// TwinCAT 3 PLC project BROTLib
// Title: BROTLib
// Company: BROT
// ProjectVersion: 0.6.1
// ProgramVersion: 3.1.4026.16
// libraries:
//   AstroBROT, * (BROT)
//   Tc2_Math, * (Beckhoff Automation GmbH)
//   Tc2_MC2, * (Beckhoff Automation GmbH)
//   Tc2_MC2_Drive, * (Beckhoff Automation GmbH)
//   Tc2_NC, * (Beckhoff Automation GmbH)
//   Tc2_Standard, * (Beckhoff Automation GmbH)
//   Tc2_System, * (Beckhoff Automation GmbH)
//   Tc2_Utilities, * (Beckhoff Automation GmbH)
//   Tc3_IotBase, * (Beckhoff Automation GmbH)
//   Tc3_IotCommunicator, * (Beckhoff Automation GmbH)
// project tree:
//   Interfaces/ I_AltAzTelescope.TcIO, I_Axis.TcIO, I_BaseAxis.TcIO, I_Brake.TcIO, I_Dome.TcIO, I_Filter.TcIO, I_Focus.TcIO, I_Hydraulics.TcIO, I_MirrorCovers.TcIO, I_Nasmyth.TcIO, I_RaDecTelescope.TcIO (not stored), I_Roof.TcIO, I_Telescope.TcIO
//   DUTs/ E_Blink.TcDUT, E_DomeRotationState.TcDUT, E_Horn.TcDUT, E_RoofState.TcDUT, E_TCSCommand.TcDUT, E_TelescopeMode.TcDUT, ST_AltAzCoordinate.TcDUT, ST_InfoDataConnection.TcDUT (not stored), ST_InfoDataFB.TcDUT (not stored), ST_InfoDataGroup.TcDUT (not stored), ST_RaDecCoordinate.TcDUT
//   GVLs/ GVL_Math.TcGVL, Global_Version.TcGVL
//   POUs/Comm/ FB_Comm_MQTT.TcPOU, FB_Comm_MQTT_Influx.TcPOU, F_EscapeInfluxString.TcPOU, F_EscapeInfluxTag.TcPOU, F_InfluxFieldValue.TcPOU, F_InfluxTimestamp.TcPOU, F_IsNumericValue.TcPOU, F_TruncateInfluxEscaped.TcPOU, I_Comm.TcIO
//   POUs/Debug/ FB_InfoConnection.TcPOU, FB_InfoEStop.TcPOU, FB_InfoGroup.TcPOU
//   POUs/ FB_AstroClock.TcPOU, FB_AstroClockSync.TcPOU, F_SetpointEnableExecute.TcPOU, FB_Axis.TcPOU, FB_BaseAxis.TcPOU, FB_BLINK.TcPOU, FB_ButtonEnable.TcPOU, FB_EventLog.TcPOU, FB_Horn.TcPOU, FB_InfluxMessage.TcPOU, FB_TONTP.TcPOU, F_YREAL.TcPOU, NCError_TO_STRING.TcPOU
//   POUs/Pointing/ FB_PointingModelForward.TcPOU, FB_PointingModelInversion.TcPOU
//   POUs/Tracking/ F_Azimuthvelocity.TcPOU, F_DerotatorPosition2.TcPOU, F_Derotatorvelocity.TcPOU, F_Elevationvelocity.TcPOU
//   Telescope/ FB_AltAzTelescopeControl.TcPOU, FB_BaseTelescopeControl.TcPOU, FB_RaDecTelescopeControl.TcPOU, ST_TelescopeConfig.TcDUT

// ---- DUTs/E_Blink.TcDUT
{attribute 'qualified_only'}
{attribute 'strict'}
TYPE E_Blink :
(
	off := 0,
	slow,
	fast,
	short,
	long,
	on
);
END_TYPE

// ---- DUTs/E_DomeRotationState.TcDUT
{attribute 'qualified_only'}
{attribute 'strict'}
TYPE E_DomeRotationState :
(
	idle  := 0,
	parked	:= 1,
	slewing := 2,
	error	:= 3,
	unknown := 4
);
END_TYPE

// ---- DUTs/E_Horn.TcDUT
{attribute 'qualified_only'}
{attribute 'strict'}
TYPE E_Horn :
(
	off := 0,
	beep,
	short,
	long
);
END_TYPE

// ---- DUTs/E_RoofState.TcDUT
{attribute 'qualified_only'}
{attribute 'strict'}
TYPE E_RoofState :
(
	closed := 0,
	opened := 1,
	opening := 2,
	closing := 3,
	stopped := 4,
	error := 5,
	unknown := 6
);
END_TYPE

// ---- DUTs/E_TCSCommand.TcDUT
{attribute 'qualified_only'}
{attribute 'strict'}
TYPE E_TCSCommand :
(
	no_command := 0,
	gohome,
	park,
	track,
	goto,
	stop,
	slew,
	poweron
);
END_TYPE

// ---- DUTs/E_TelescopeMode.TcDUT
{attribute 'qualified_only'}
{attribute 'strict'}
TYPE E_TelescopeMode :
(
	off := 0,
	manual := 1,
	automatic := 2
);
END_TYPE

// ---- DUTs/ST_AltAzCoordinate.TcDUT
TYPE ST_AltAzCoordinate :
STRUCT
	Altitude : LREAL;
	Azimuth  : LREAL;
END_STRUCT
END_TYPE

// ---- DUTs/ST_RaDecCoordinate.TcDUT
TYPE ST_RaDecCoordinate :
STRUCT
	RightAscension  : LREAL;
	Declination : LREAL;
END_STRUCT
END_TYPE

// ---- Telescope/ST_TelescopeConfig.TcDUT
TYPE ST_TelescopeConfig :
STRUCT
	// location
	longitude			: LREAL; // telescope site longitude
	latitude			: LREAL; // telescope site latitude
	altitude			: LREAL; // telescope site height above sea level: estimated
	
	// park position
	elevationPark		: LREAL;
	azimuthPark			: LREAL;
	derotatorPark		: LREAL;
	focusPark			: LREAL;

	// home position
	elevationHome		: LREAL;
	azimuthHome			: LREAL;
	derotatorHome		: LREAL;
	
	// information about telescope
	name				: STRING;
	diameter			: LREAL;
	cabinet				: STRING;
	manufacturer		: STRING;
	
	// and about the mount
	mountOptions		: STRING;
	mount				: STRING;	
END_STRUCT
END_TYPE

// ---- GVLs/GVL_Math.TcGVL
{attribute 'qualified_only'}
VAR_GLOBAL CONSTANT
	LREAL_MIN			: LREAL :=  -1.7976931348623157E+308; // https://infosys.beckhoff.com/index.php?content=../content/1031/tc3_plc_intro/2529405067.html&id=
	// literal values (PI/180 and 180/PI), not PI-based expressions: PI is not initialised yet when these
	// constants are, which fails the build ("uninitialized variable PI is used for initialization")
	d2r					: LREAL := 0.017453292519943295;
	r2d					: LREAL := 57.29577951308232;
	// Earth's mean sidereal angular rate, deg/s (360 deg / 86164.0905 s mean sidereal day); was previously
	// copy-pasted into three tracking functions, and separately (re-derived slightly differently, as
	// 360/86164.099, ~0.005 arcsec/hour off) as the unused FB_BaseTelescopeControl.fSiderialVelocity
	Omega				: LREAL := 4.178074605556E-3;
END_VAR

// ---- GVLs/Global_Version.TcGVL
{attribute 'qualified_only'}
VAR_GLOBAL CONSTANT
	// Mirrors Beckhoff's own Global_Version.stLibVersion_* pattern (see ST_LibVersion),
	// which only covers Tc2_*/Tc3_* library references, not custom ones -- until now: this
	// GVL uses Beckhoff's own naming exactly, so it merges into a consumer's Global_Version.
	// Kept in sync with <ProjectVersion> in BROTLib.plcproj at release time.
	stLibVersion_BROTLib : ST_LibVersion := (
		iMajor := 0,
		iMinor := 6,
		iBuild := 1,
		iRevision := 0,
		nFlags := 1,
		sVersion := '0.6.1'
	);
END_VAR

// ---- Interfaces/I_AltAzTelescope.TcIO
INTERFACE I_AltAzTelescope EXTENDS I_Telescope

PROPERTY AltitudeOffset : LREAL
GET
END_GET
SET
END_SET
END_PROPERTY

PROPERTY AzimuthOffset : LREAL
GET
END_GET
SET
END_SET
END_PROPERTY

PROPERTY DerotatorOffset : LREAL
GET
END_GET
SET
END_SET
END_PROPERTY

PROPERTY Dut1 : LREAL
GET
END_GET
SET
END_SET
END_PROPERTY

END_INTERFACE

// ---- Interfaces/I_Axis.TcIO
INTERFACE I_Axis EXTENDS I_BaseAxis

PROPERTY ActualPosition : LREAL
GET
END_GET
SET
END_SET
END_PROPERTY

PROPERTY isTracking : BOOL
GET
END_GET
END_PROPERTY

PROPERTY MoveAxis : BOOL
GET
END_GET
SET
END_SET
END_PROPERTY

PROPERTY MoveDone : BOOL
GET
END_GET
END_PROPERTY

PROPERTY SlewTime : LREAL
GET
END_GET
END_PROPERTY

PROPERTY StopAxis : BOOL
GET
END_GET
SET
END_SET
END_PROPERTY

PROPERTY Tracking : BOOL
GET
END_GET
SET
END_SET
END_PROPERTY

END_INTERFACE

// ---- Interfaces/I_BaseAxis.TcIO
INTERFACE I_BaseAxis

PROPERTY ActualPosition : LREAL
GET
END_GET
SET
END_SET
END_PROPERTY

PROPERTY Busy : BOOL
GET
END_GET
END_PROPERTY

PROPERTY Calibrated : BOOL
GET
END_GET
END_PROPERTY

PROPERTY Enable : BOOL
GET
END_GET
SET
END_SET
END_PROPERTY

PROPERTY Error : BOOL
GET
END_GET
END_PROPERTY

PROPERTY ErrorID : UDINT
GET
END_GET
END_PROPERTY

PROPERTY HomeAxis : BOOL
GET
END_GET
SET
END_SET
END_PROPERTY

PROPERTY InNegLimit : BOOL
GET
END_GET
END_PROPERTY

PROPERTY InPosLimit : BOOL
GET
END_GET
END_PROPERTY

PROPERTY MoveNeg : BOOL
GET
END_GET
SET
END_SET
END_PROPERTY

PROPERTY MovePos : BOOL
GET
END_GET
SET
END_SET
END_PROPERTY

PROPERTY Position : LREAL
GET
END_GET
SET
END_SET
END_PROPERTY

PROPERTY Ready : BOOL
GET
END_GET
END_PROPERTY

METHOD Reset : BOOL
VAR_INPUT
END_VAR
END_METHOD

PROPERTY Velocity : LREAL
GET
END_GET
SET
END_SET
END_PROPERTY

END_INTERFACE

// ---- Interfaces/I_Brake.TcIO
INTERFACE I_Brake

PROPERTY BrakeOpen : BOOL
GET
END_GET
END_PROPERTY

METHOD CloseBrake : BOOL
VAR_INPUT
END_VAR
END_METHOD

METHOD OpenBrake : BOOL
VAR_INPUT
END_VAR
END_METHOD

END_INTERFACE

// ---- Interfaces/I_Dome.TcIO
INTERFACE I_Dome

PROPERTY Capabilities : INT
GET
END_GET
END_PROPERTY

METHOD Close : BOOL
VAR_INPUT
END_VAR
END_METHOD

PROPERTY Error : BOOL
GET
END_GET
END_PROPERTY

PROPERTY ErrorID : UDINT
GET
END_GET
END_PROPERTY

METHOD Open : BOOL
VAR_INPUT
END_VAR
END_METHOD

METHOD Park : BOOL
VAR_INPUT
END_VAR
END_METHOD

PROPERTY Parked : BOOL
GET
END_GET
END_PROPERTY

PROPERTY Position : LREAL
GET
END_GET
SET
END_SET
END_PROPERTY

METHOD Reset : BOOL
VAR_INPUT
END_VAR
END_METHOD

PROPERTY RotState : E_DomeRotationState
GET
END_GET
END_PROPERTY

PROPERTY ShutterState : E_RoofState
GET
END_GET
SET
END_SET
END_PROPERTY

METHOD Stop : BOOL
VAR_INPUT
END_VAR
END_METHOD

METHOD StopTrack : BOOL
VAR_INPUT
END_VAR
END_METHOD

METHOD Track : BOOL
VAR_INPUT
END_VAR
END_METHOD

PROPERTY Tracking : BOOL
GET
END_GET
END_PROPERTY

END_INTERFACE

// ---- Interfaces/I_Filter.TcIO
INTERFACE I_Filter

METHOD SetFilter : BOOL
VAR_INPUT
	FilterPos	: USINT;
END_VAR
END_METHOD

END_INTERFACE

// ---- Interfaces/I_Focus.TcIO
INTERFACE I_Focus EXTENDS I_BaseAxis

END_INTERFACE

// ---- Interfaces/I_Hydraulics.TcIO
INTERFACE I_Hydraulics

PROPERTY Enable : BOOL
GET
END_GET
SET
END_SET
END_PROPERTY

PROPERTY Error : BOOL
GET
END_GET
END_PROPERTY

PROPERTY ManualStartSuction : BOOL
GET
END_GET
SET
END_SET
END_PROPERTY

PROPERTY ManualStopPump : BOOL
GET
END_GET
SET
END_SET
END_PROPERTY

PROPERTY OilPressureOK : BOOL
GET
END_GET
END_PROPERTY

PROPERTY PumpRunning : BOOL
GET
END_GET
END_PROPERTY

METHOD Reset : BOOL
VAR_INPUT
END_VAR
END_METHOD

PROPERTY SuctionRunning : BOOL
GET
END_GET
END_PROPERTY

END_INTERFACE

// ---- Interfaces/I_MirrorCovers.TcIO
INTERFACE I_MirrorCovers

METHOD Close : BOOL
VAR_INPUT
END_VAR
END_METHOD

PROPERTY Closed : BOOL
GET
END_GET
END_PROPERTY

PROPERTY Error : BOOL
GET
END_GET
END_PROPERTY

METHOD Open : BOOL
VAR_INPUT
END_VAR
END_METHOD

PROPERTY Opened : BOOL
GET
END_GET
END_PROPERTY

METHOD Reset : BOOL
VAR_INPUT
END_VAR
END_METHOD

END_INTERFACE

// ---- Interfaces/I_Nasmyth.TcIO
INTERFACE I_Nasmyth

METHOD SetNasmyth : BOOL
VAR_INPUT
	Port	: INT;
END_VAR
END_METHOD

END_INTERFACE

// ---- Interfaces/I_Roof.TcIO
INTERFACE I_Roof

METHOD Close : BOOL
VAR_INPUT
END_VAR
END_METHOD

METHOD Open : BOOL
VAR_INPUT
END_VAR
END_METHOD

METHOD Reset : BOOL
VAR_INPUT
END_VAR
END_METHOD

PROPERTY State : E_RoofState
GET
END_GET
END_PROPERTY

METHOD Stop : BOOL
VAR_INPUT
END_VAR
END_METHOD

END_INTERFACE

// ---- Interfaces/I_Telescope.TcIO
INTERFACE I_Telescope

PROPERTY Altitude : LREAL
GET
END_GET
END_PROPERTY

PROPERTY Azimuth : LREAL
GET
END_GET
END_PROPERTY

PROPERTY CoverAutoOpen : BOOL
GET
END_GET
SET
END_SET
END_PROPERTY

PROPERTY Declination : LREAL
GET
END_GET
END_PROPERTY

METHOD ABSTRACT Home : BOOL
VAR_INPUT
END_VAR
END_METHOD

METHOD Init : BOOL
VAR_INPUT
END_VAR
END_METHOD

METHOD ABSTRACT Park : BOOL
VAR_INPUT
END_VAR
END_METHOD

METHOD Reset : BOOL
VAR_INPUT
END_VAR
END_METHOD

PROPERTY RightAscension : LREAL
GET
END_GET
END_PROPERTY

METHOD Slew : BOOL
VAR_INPUT
	fAzimuth		: LREAL;
	fAltitude		: LREAL;
END_VAR
END_METHOD

METHOD Stop : BOOL
VAR_INPUT
END_VAR
END_METHOD

METHOD Track : BOOL
VAR_INPUT
	fRightAscension	: LREAL;
	fDeclination	: LREAL;
END_VAR
END_METHOD

END_INTERFACE

// ---- POUs/Comm/I_Comm.TcIO
INTERFACE I_Comm

METHOD Publish : BOOL
VAR_INPUT
	domain			: STRING(255) := 'environment';
	location		: STRING(255) := 'roof';
	parameter		: STRING(255);
	value			: STRING(255);	
END_VAR
VAR_OUTPUT
	published	: BOOL;
END_VAR
END_METHOD

METHOD PublishLog : BOOL
VAR_INPUT
	level		: STRING(255) := 'INFO';
	message		: STRING(255);	
END_VAR
VAR_OUTPUT
	published	: BOOL;
END_VAR
END_METHOD

END_INTERFACE

// ---- Telescope/FB_BaseTelescopeControl.TcPOU
FUNCTION_BLOCK ABSTRACT FB_BaseTelescopeControl IMPLEMENTS I_Telescope
VAR_INPUT
(*
TCS interface section, modeled on an external TCS spec kept as a private internal reference
(not linked here -- this repo is public; ask internally for the spec if you need it). See
specs/design/telescope-telemetry-publish-chain.md for what's actually confirmed about the
on-wire format from tracing the code, since the spec itself isn't accessible from here.
*)
	bPower				: BOOL;		// true: Power on
	bGoHome				: BOOL;		// true: go to home position, unset track/goto if active
	bPark				: BOOL;		// boolean, true: go into park position, ready to stow telescope, unset track/goto
	bTrack				: BOOL;		// boolean, TRUE: MOVE telescope TO last ra/de AND start tracking. Set 'goto' TO FALSE, IF TRUE. FALSE: Stop tracking as soon as possible
	bGoto				: BOOL;		// boolean, TRUE: MOVE telescope TO tau/de AND stop there. Set track TO FALSE, IF TRUE. FALSE: no effect.)	
	bSlew				: BOOL;		// move the telescope to a given az-alt position
	bStop				: BOOL;		// boolean, TRUE: Stop motion OF telescope immediately, set goto AND track TO FALSE. FALSE: Allow motion OF telescope again via track/goto).	
	bReset				: BOOL;		// initiates reset on all axis
	bAutoTrack			: BOOL := TRUE;	// automatic tracking after goto
	bCoverAutoOpen		: BOOL := TRUE;	// automatically open the mirror covers on Init/PowerOn
	// catalog/mean right ascension (ICRS/J2000), degrees, double -- fed straight into AstroBROT's
	// FB_EQ2HOR with precess/nutate/aberration all at their default TRUE, which only makes sense
	// for mean/catalog input (feeding it an already-apparent position would double-correct it);
	// MONETcommon's own telemetry independently re-publishes this same value as *_RA_ICRS (#22)
	fRightAscension		: LREAL :=  0.0;
	// catalog/mean declination (ICRS/J2000), degrees, double -- see fRightAscension
	fDeclination		: LREAL :=  0.0;
	fElevation			: LREAL :=  0.0;	// desired elevation of the telescope pointing
	fAzimuth			: LREAL :=  0.0;	// desired azimut of the telescope pointing
	fTimeOffset			: LREAL := 0.0;		// absolute offset for time
	fHorizon			: LREAL := 1.0;		// ELEVATION below which value the telescope will not go
	
	// TRUE while the E-stop is triggered. The caller must connect it to its safety handling (MONETS/MONETN MAIN:
	// SafetyHandling.estop); left unconnected, the E-stop is never reported as STATUS.GLOBAL = 1 (#10).
	bEstopTriggered		: BOOL	:= FALSE;
	bMainReady			: BOOL	:= TRUE;
	
	telescopeConfig		: ST_TelescopeConfig;
END_VAR
VAR
	fbComm 				: I_Comm;
	
	TCS_command			: E_TCSCommand;	// actual command from the TCS
	// fJd/fLst are published by _PublishTelemetry, but this block never sets them or calls fbTime: the derived
	// block must (MONETcommon's FB_MonetTelescopeControl does, gated on fbTime.bValid). Otherwise both read 0 (#10).
	fJd					: LREAL;	// current Julian Date calculated from system time
	fLst				: LREAL;	// local siderial time calculated from Julian date in hours
	fElevationCalc		: LREAL;	// elevation calulated when ra and dec are set by TCS 
	fAzimuthCalc		: LREAL;	// azimuth calulated when ra and dec are set by TCS
	fHourAngle			: LREAL;	// hourangle when ra and dec are set by TCS
	
	fRightAscensionCalc	: LREAL;	// right ascension calulated when azimuth and elevation are set by TCS
	fDeclinationCalc	: LREAL;	// declination calulated when azimuth and elevation are set by TCS
	fHourAngleCalc		: LREAL;	// hour angle azimuth and elevation are set by TCS
	
	fbTime				: FB_AstroClock;	// precise astronomical	time
	
	rtrigReset			: R_TRIG;
	bInterrupted		: BOOL;		// If a command is interruped by one with more presedence, the interrupted needs to reset its stage
	
	bPowerFailure		: BOOL;		// triggers power-failure event
	tpPowerOnWarning	: TP;		// triggers power warning
	tonPowerTimeout		: TON;		// power on timeout
	tonCommandTimeout	: TON;		// command timeout
	tonTrackingDelay	: TON;		// tracking delay
	
	TCSpowerEvent,
	TCSgohomeEvent,
	TCSparkEvent,
	TCSgotoEvent,
	TCStrackEvent,
	TCSstopEvent,
	TCStargetHorizonEvent,
	TCSaltitudeEvent,
	TCSnearPoleEvent,
	TCSreadyEvent,
	TCSCTOEvent			: FB_Eventlog;
	tonMQTTTimer 			: TON := (PT:=T#5S);
	// the 7 INFO/CONFIG fields never change at runtime; republishing them on the fast 1-5s
	// telemetry cadence is wasted traffic, so they get their own much slower timer instead
	tonStaticTelemetryTimer	: TON := (PT:=T#30S);
	bStaticTelemetrySent	: BOOL;	// forces one immediate publish on the first cycle
END_VAR
VAR_OUTPUT
	bReady				: BOOL;		// TRUE, IF telescope can be operated 
	fReadyState 		: LREAL := 0.0; // 0: Shut down, 1 powered on, -1 Error
	bIsParked			: BOOL := TRUE;		// telescope is parked
	bIsPowered			: BOOL;		// telescope is powered on
	bError				: BOOL;		// indicates an error on one of the components
	bHorizonError		: BOOL;		// if TRUE, the set Coordinate is below the Horizon threshold fHorizon
	nErrorID				: UDINT;	//error id of axis
	nMotionState		: INT	:= 0;
	bSlewing			: BOOL;		//TRUE, IF telescope is in fast-MOVE phase (includes pole-swap)	
	bTracking			: BOOL;		//TRUE, IF telescope is on tracking position AND currently tracking.	
	bStopped			: BOOL;		//TRUE, IF telescope is AT rest.	
	fHourAngleCurrent	: LREAL;	// true position of the hour angle (without pointing and offset correction)
	fDeclinationCurrent	: LREAL;	// true position of the declination (without pointing and offset correction)
	fRightAscensionCurrent: LREAL;	// true position of the right ascension (without pointing and offset correction)
	fElevationCurrent	: LREAL;	// current position in elevation (calculated) (without pointing and offset correction)
	fAzimuthCurrent		: LREAL;	// current position in azimuth (calculated) (without pointing and offset correction)
	fElevationCurrentSky	: LREAL;	// current position in elevation (calculated)
	fAzimuthCurrentSky		: LREAL;	// current position in azimuth (calculated)
	fSlewTime			: LREAL;	//	(time in sec. to reach the goto/track position) 
	bHomed				: BOOL;		// True: telescope is calibrated
	bBusy				: BOOL;		// telescope does not accept further commands
END_VAR
VAR CONSTANT
	// kept as an inherited constant (not GVL_Math.d2r directly) so existing subclasses
	// (e.g. MONETcommon/MONETN's FB_MonetTelescopeControl) keep working unmodified; single-sourced
	// from GVL_Math now instead of its own copy of PI/180.0
	d2r		: LREAL := GVL_Math.d2r;
END_VAR


// telemetry cadence depends on state: every 1s while slewing/tracking, every 5s otherwise
// (subclasses that don't call SUPER^() from their own cyclic body, e.g. MONETcommon's
// FB_MonetTelescopeControl, drive this on their own timer instead and call _PublishTelemetry()
// directly -- the static-fields gating below lives inside that method, not here, so it still
// applies either way)
IF bSlewing OR bTracking THEN
	tonMQTTTimer.PT := T#1000MS;
ELSE
	tonMQTTTimer.PT := T#5000MS;
END_IF
tonMQTTTimer(IN:=TRUE);
IF tonMQTTTimer.Q THEN
	tonMQTTTimer(IN:=FALSE);
	_PublishTelemetry();
END_IF

METHOD _PublishTelemetry : BOOL
VAR_INPUT
END_VAR
// fbComm is only ever set via FB_Init(comm := ...); nothing enforces that a consumer actually
// does, and calling through an unassigned interface reference crashes the whole PLC task (#7)
IF fbComm = 0 THEN
	RETURN;
END_IF

(* TELESCOPE module*)

//fbComm.Publish('telescope', 'dome', 'TELESCOPE.READY_STATE',	LREAL_TO_STRING(fReadyState));
//fbComm.Publish('telescope', 'dome', 'TELESCOPE.Motion_STATE',	LREAL_TO_STRING(nMotionState));

// static INFO/CONFIG fields never change at runtime: publish once immediately, then only every
// 30s afterward, instead of on every call to this method (#22). Gated here rather than in the
// cyclic body so it still applies when a subclass calls this method directly on its own timer
// instead of going through FB_BaseTelescopeControl's own cyclic body (e.g. MONETcommon's
// FB_MonetTelescopeControl, which never calls SUPER^() from its main body)
tonStaticTelemetryTimer(IN:=TRUE);
IF NOT bStaticTelemetrySent OR tonStaticTelemetryTimer.Q THEN
	tonStaticTelemetryTimer(IN:=FALSE);
	bStaticTelemetrySent := TRUE;
	_PublishStaticTelemetry();
END_IF

// STATUS
IF bEstopTriggered THEN
	fbComm.Publish('telescope', 'dome', 'TELESCOPE.STATUS.GLOBAL', '1');
ELSIF bError THEN
	fbComm.Publish('telescope', 'dome', 'TELESCOPE.STATUS.GLOBAL', '2');
ELSE
	fbComm.Publish('telescope', 'dome', 'TELESCOPE.STATUS.GLOBAL', '0');
END_IF
(* ERROR LIST: TO BE IMPLEMENTED!!!*)

(* OBJECT Module*)

// INSTRUMENTAL
// Set Coords from outside | GoTo:RA DEC | Slew:Alt Az
fbComm.Publish('telescope', 'dome', 'OBJECT.INSTRUMENTAL.RA', LREAL_TO_STRING(fRightAscension));
fbComm.Publish('telescope', 'dome', 'OBJECT.INSTRUMENTAL.DEC', LREAL_TO_STRING(fDeclination));
fbComm.Publish('telescope', 'dome', 'OBJECT.INSTRUMENTAL.ALT', LREAL_TO_STRING(fElevation));
fbComm.Publish('telescope', 'dome', 'OBJECT.INSTRUMENTAL.AZ', LREAL_TO_STRING(fAzimuth));

// HORIZONTAL
IF bSlew THEN
	fbComm.Publish('telescope', 'dome', 'OBJECT.HORIZONTAL.ALT', LREAL_TO_STRING(fElevation));
	fbComm.Publish('telescope', 'dome', 'OBJECT.HORIZONTAL.AZ', LREAL_TO_STRING(fAzimuth));
ELSE
	fbComm.Publish('telescope', 'dome', 'OBJECT.HORIZONTAL.ALT', LREAL_TO_STRING(fElevationCalc));
	fbComm.Publish('telescope', 'dome', 'OBJECT.HORIZONTAL.AZ', LREAL_TO_STRING(fAzimuthCalc));
END_IF

//EQUATORIAL
fbComm.Publish('telescope', 'dome', 'OBJECT.EQUATORIAL.EPOCH', 'J2000.0');
fbComm.Publish('telescope', 'dome', 'OBJECT.EQUATORIAL.EQUINOX', 'J2000.0');
fbComm.Publish('telescope', 'dome', 'OBJECT.EQUATORIAL.RA_PM', '0.0');
fbComm.Publish('telescope', 'dome', 'OBJECT.EQUATORIAL.DEC_PM', '0.0');
fbComm.Publish('telescope', 'dome', 'OBJECT.EQUATORIAL.RA_RATE', '0.0');
fbComm.Publish('telescope', 'dome', 'OBJECT.EQUATORIAL.DEC_RATE', '0.0');
// all angles in the telemetry are degrees, RA included, like the rightascension command (#37)
IF bSlew THEN
	fbComm.Publish('telescope', 'dome', 'OBJECT.EQUATORIAL.RA', LREAL_TO_STRING(fRightAscensionCalc));
	fbComm.Publish('telescope', 'dome', 'OBJECT.EQUATORIAL.DEC', LREAL_TO_STRING(fDeclinationCalc));
ELSE
	fbComm.Publish('telescope', 'dome', 'OBJECT.EQUATORIAL.RA', LREAL_TO_STRING(fRightAscension));
	fbComm.Publish('telescope', 'dome', 'OBJECT.EQUATORIAL.DEC', LREAL_TO_STRING(fDeclination));
END_IF

(*POSITION*)
//LOCAL
fbComm.Publish('telescope', 'dome', 'POSITION.LOCAL.SIDEREAL_TIME', LREAL_TO_STRING(fLst));
fbComm.Publish('telescope', 'dome', 'POSITION.LOCAL.JD', LREAL_TO_STRING(fJd));
fbComm.Publish('telescope', 'dome', 'POSITION.LOCAL.LATITUDE', LREAL_TO_STRING(telescopeConfig.latitude));
fbComm.Publish('telescope', 'dome', 'POSITION.LOCAL.LONGITUDE', LREAL_TO_STRING(telescopeConfig.longitude));
fbComm.Publish('telescope', 'dome', 'POSITION.LOCAL.HEIGHT', LREAL_TO_STRING(telescopeConfig.altitude));
END_METHOD

METHOD _PublishStaticTelemetry : BOOL
VAR_INPUT
END_VAR
// see _PublishTelemetry's identical guard (#7)
IF fbComm = 0 THEN
	RETURN;
END_IF

// fields that never change at runtime -- published on their own slow timer (see the cyclic
// body), not on _PublishTelemetry's fast 1-5s cadence (#22)

// INFO
fbComm.Publish('telescope', 'dome', 'TELESCOPE.INFO.NAME',	telescopeConfig.name);
fbComm.Publish('telescope', 'dome', 'TELESCOPE.INFO.DIAMETER',	LREAL_TO_STRING(telescopeConfig.diameter));
fbComm.Publish('telescope', 'dome', 'TELESCOPE.INFO.CABINET',	telescopeConfig.cabinet);
fbComm.Publish('telescope', 'dome', 'TELESCOPE.INFO.MANUFACTURER', telescopeConfig.manufacturer);

// CONFIG
fbComm.Publish('telescope', 'dome', 'TELESCOPE.CONFIG.CAPABILITIES', '0'); // no ST_TelescopeConfig field for this yet
fbComm.Publish('telescope', 'dome', 'TELESCOPE.CONFIG.MOUNTOPTIONS', telescopeConfig.mountOptions);
fbComm.Publish('telescope', 'dome', 'TELESCOPE.CONFIG.MOUNT', telescopeConfig.mount);
END_METHOD

PROPERTY Altitude : LREAL
GET
Altitude := THIS^.fElevationCurrent;
END_GET
END_PROPERTY

PROPERTY Azimuth : LREAL
GET
Azimuth := THIS^.fAzimuthCurrent;
END_GET
END_PROPERTY

PROPERTY CoverAutoOpen : BOOL
GET
CoverAutoOpen := THIS^.bCoverAutoOpen;
END_GET
SET
THIS^.bCoverAutoOpen := CoverAutoOpen;
END_SET
END_PROPERTY

PROPERTY Declination : LREAL
GET
Declination := THIS^.fDeclinationCurrent;
END_GET
END_PROPERTY

METHOD FB_init : BOOL
VAR_INPUT
	bInitRetains : BOOL; // if TRUE, the retain variables are initialized (warm start / cold start)
	bInCopyCode : BOOL;  // if TRUE, the instance afterwards gets moved into the copy code (online change)
	comm			: I_Comm;	
END_VAR
THIS^.fbComm := comm;
END_METHOD

METHOD Home : BOOL
bGoHome := TRUE;
END_METHOD

METHOD Init : BOOL
bPower := TRUE;
END_METHOD

METHOD Park : BOOL
bPark := TRUE;
END_METHOD

METHOD Reset : BOOL
VAR_INPUT
END_VAR
bReset := TRUE;
END_METHOD

PROPERTY RightAscension : LREAL
GET
RightAscension := THIS^.fRightAscensionCurrent;
END_GET
END_PROPERTY

METHOD Slew : BOOL
VAR_INPUT
	fAzimuth		: LREAL;
	fAltitude		: LREAL;
END_VAR
THIS^.fAzimuth := fAzimuth;
THIS^.fElevation := fAltitude;
bSlew := TRUE;
END_METHOD

METHOD Stop : BOOL
bStop := TRUE;
END_METHOD

METHOD Track : BOOL
VAR_INPUT
	fRightAscension	: LREAL;
	fDeclination	: LREAL;
END_VAR
THIS^.fRightAscension := fRightAscension;
THIS^.fDeclination := fDeclination;
bTrack := TRUE;
END_METHOD

END_FUNCTION_BLOCK

// ---- POUs/FB_AstroClock.TcPOU
// Software clock (RTC_EX2, microsecond resolution) resynchronised from the Windows system time every 5 s.
// NT_GetTime returns the LOCAL Windows time and nothing here converts it, so the PLC's Windows time zone must be
// UTC: DateTime2JD and everything downstream (LST, pointing, tracking) expect UTC. The production PCs are set to UTC.
// Check bValid before using time_RTCEX2 (see FB_AstroClockSync).
FUNCTION_BLOCK FB_AstroClock
VAR_INPUT
END_VAR
VAR_OUTPUT
        bValid          : BOOL;         // FALSE until the first successful sync; stays TRUE afterwards, the RTC keeps counting
        nSyncErrors     : UINT;         // failed syncs in a row (diagnostics)
        time_RTCEX2     : TIMESTRUCT;
        nMicroseconds   : DWORD;
END_VAR
VAR
	        fbGetLocalTime  : NT_GetTime;
        bBusy           : BOOL;
        bError          : BOOL;
        nErrID          : UDINT;
        presetTime      : TIMESTRUCT;

        syncTimer       : TON;
        fbSync          : FB_AstroClockSync;
        bSynchronize    : BOOL;

        fbRTC_EX2       : RTC_EX2;
        bValid_RTCEX2   : BOOL;
END_VAR

(*
TYPE TIMESTRUCT
STRUCT
   wYear            : WORD;
   wMonth           : WORD;
   wDayOfWeek       : WORD;
   wDay             : WORD;
   wHour            : WORD;
   wMinute          : WORD;
   wSecond          : WORD;
   wMilliseconds    : WORD;
END_STRUCT
END_TYPE
*)

syncTimer(IN := NOT SyncTimer.Q, PT := T#5S);
fbGetLocalTime(START := syncTimer.Q,
	TMOUT := DEFAULT_ADS_TIMEOUT,
	Busy => bBusy,
	ERR => bError,
	ERRID => nErrID,
	TIMESTR => presetTime);

// the RTC is loaded only after a successful read; bValid tells callers whether time_RTCEX2 can be used
fbSync(bBusy := bBusy, bError := bError,
	bSynchronize => bSynchronize,
	bValid => bValid,
	nErrors => nSyncErrors);

fbRTC_EX2(EN := bSynchronize,
	PDT := presetTime,
	PMICRO := 0,
	Q => bValid_RTCEX2,
	CDT => time_RTCEX2,
	CMICRO => nMicroseconds);

END_FUNCTION_BLOCK

// ---- POUs/FB_AstroClockSync.TcPOU
// Decides when FB_AstroClock may load the RTC blocks and whether the time can be trusted.
// Separate from FB_AstroClock so that it runs without ADS and can be unit tested.
//
// Feed it the Busy and Err outputs of NT_GetTime. The decision is taken at the moment Busy falls, because
// NT_GetTime raises Err in the same cycle: bSynchronize pulses for one cycle after a successful read only.
// A failed read must not load the RTCs, because the time structure it returns is stale (zero on the first call).
FUNCTION_BLOCK FB_AstroClockSync
VAR_INPUT
	bBusy			: BOOL;				// NT_GetTime.Busy
	bError			: BOOL;				// NT_GetTime.Err
END_VAR
VAR_OUTPUT
	bSynchronize	: BOOL;				// one cycle: load the RTCs from the time just read
	bValid			: BOOL;				// TRUE from the first successful read on; stays TRUE, the RTC keeps counting
	nErrors			: UINT;				// failed reads in a row (saturates at 65535), for diagnostics
END_VAR
VAR
	fbBusyDone		: F_TRIG;
	bEverSynchronized	: BOOL;
END_VAR

fbBusyDone(CLK := bBusy);
bSynchronize := FALSE;

IF fbBusyDone.Q THEN
	IF bError THEN
		IF nErrors < 65535 THEN
			nErrors := nErrors + 1;
		END_IF
	ELSE
		bSynchronize := TRUE;
		bEverSynchronized := TRUE;
		nErrors := 0;
	END_IF
END_IF

// After the first sync the RTC keeps counting on its own, so failed reads only make the last sync older (drift is
// far below a second over minutes). Only the time before the first sync is garbage, so that is all bValid excludes.
bValid := bEverSynchronized;

END_FUNCTION_BLOCK

// ---- POUs/FB_EventLog.TcPOU
FUNCTION_BLOCK FB_EventLog
VAR_INPUT
	Trigger			: BOOL;
	// ADSLOG_MSGTYPE_HINT or ADSLOG_MSGTYPE_WARN or ADSLOG_MSGTYPE_ERROR
	Level			: UDINT := ADSLOG_MSGTYPE_HINT;
	FormatString	: STRING(255) := '%s';
	OnMessage		: STRING(255) := '';
	OffMessage		: STRING(255) := '';
	OffLevel		: UDINT := ADSLOG_MSGTYPE_HINT;
	Comm			: I_Comm;
END_VAR
VAR_OUTPUT
END_VAR
VAR
	LogonTrigger	: R_TRIG;
	LogoffTrigger	: F_TRIG; // R_Trig or F_Trig ?!
	PayloadMessage	: STRING(255);
	fbFormat		: FB_FormatString;
	// OffLevel is a VAR_INPUT; fall back to Level in a local instead of writing back into it
	effectiveOffLevel	: UDINT;
END_VAR

LogonTrigger(CLK := Trigger);
LogoffTrigger(CLK := Trigger);
// in case the OffLevel is not set use the default Level Value
effectiveOffLevel := OffLevel;
IF effectiveOffLevel = 0 THEN
	effectiveOffLevel := Level;
END_IF
IF LogonTrigger.Q AND LEN(OnMessage)>0 THEN
	ADSLOGSTR( Level OR ADSLOG_MSGTYPE_LOG, FormatString, OnMessage);
END_IF

IF LogoffTrigger.Q AND LEN(OffMessage)>0 THEN
	ADSLOGSTR( effectiveOffLevel OR ADSLOG_MSGTYPE_LOG, FormatString, OffMessage);
END_IF

// same length check as the ADS log above (>0), so a one-character message is not local-only.
// Comm <> 0: it's a plain VAR_INPUT, nothing stops a caller from leaving it unassigned, and
// calling through it would crash the whole PLC task (#7) -- the ADS log above still happens
// either way, only the MQTT publish is skipped
IF LogonTrigger.Q AND LEN(OnMessage)>0 AND Comm <> 0 THEN
	fbFormat( sFormat := FormatString, arg1 := F_STRING(OnMessage), sOut => PayloadMessage);
	Comm.PublishLog(_LevelToString(Level), PayloadMessage);
END_IF

IF LogoffTrigger.Q AND LEN(OffMessage)>0 AND Comm <> 0 THEN
	fbFormat( sFormat := FormatString, arg1 := F_STRING(OffMessage), sOut => PayloadMessage);
	Comm.PublishLog(_LevelToString(effectiveOffLevel), PayloadMessage);
END_IF

METHOD PRIVATE _LevelToString : STRING
VAR_INPUT
	level	: UDINT;
END_VAR
// bit-test rather than = against the raw constant: a caller combining Level with another flag
// (e.g. the ADSLOG_MSGTYPE_LOG bit this FB itself ORs in for ADSLOGSTR) must still match its
// actual severity here instead of always falling through to ERROR
IF (level AND ADSLOG_MSGTYPE_ERROR) <> 0 THEN
	_LevelToString := 'ERROR';
ELSIF (level AND ADSLOG_MSGTYPE_WARN) <> 0 THEN
	_LevelToString := 'WARNING';
ELSE
	_LevelToString := 'INFO';
END_IF
END_METHOD

END_FUNCTION_BLOCK

// ---- POUs/Comm/FB_Comm_MQTT.TcPOU
FUNCTION_BLOCK ABSTRACT FB_Comm_MQTT IMPLEMENTS I_Comm
VAR_INPUT
	sHostName     	: STRING(255);
    nHostPort     	: UINT := 1883;
    nKeepAlive    	: UINT := 60;
	sTopicSub    	: STRING(255);
	sTopicPublish  	: STRING(255);
	sTopicLog     	: STRING(255);
	Telescope     	: I_Telescope;
	AltAzTelescope 	: I_AltAzTelescope;
	RaDecTelescope	: I_RaDecTelescope;
	Focus			: I_Focus;
	Filter			: I_Filter;
	Nasmyth			: I_Nasmyth;
	Dome			: I_Dome;
	Roof			: I_Roof;
	MirrorCovers	: I_MirrorCovers;
END_VAR
VAR_OUTPUT
	bConnected    	: BOOL := FALSE;
END_VAR
VAR
	state     		: INT := 0;
	GetHostName		: FB_GetHostName;
	HostName		: STRING(255);
	
	{attribute 'TcEncoding':='UTF-8'}
	sTopicRcv: 			STRING(255);
	{attribute 'TcEncoding':='UTF-8'}
	fbMessageQueue:		FB_IotMqttMessageQueue;
    fbMessage:			FB_IotMqttMessage;
	fbMqttClient:		FB_IotMqttClient;
	// match _handleMQTTMessage's sPayloadRcv : STRING(255) -- plain STRING (80 chars) here
	// truncated any longer message before it ever reached the 255-capable handler (#24)
	sPayloadRcv: 		STRING(255);
	tonHostNameStuck	: TON := (PT := T#30S);	// warn once if state 0 never completes (#5)
	bHostNameStuckLogged: BOOL;
	sStatusTopic		: STRING(255);	// {sTopicPublish}/status: 'online'/'offline' presence (#5)
	sOnlinePayload		: STRING(20);
	sOfflinePayload		: STRING(20);
END_VAR

(*
MQTT Communication section

Source:
https://infosys.beckhoff.com/english.php?content=../content/1033/tf6701_tc3_iot_communication_mqtt/3518541195.html&id=

*)

CASE state OF
0:
	// get hostname of this machine
	GetHostName(bExecute := TRUE, sHostName => HostName);

	// finished?
	IF HostName <> '' THEN
		GetHostName(bExecute := FALSE);
		state := 1;
	ELSE
		// GetHostName failing would otherwise leave this state (and the whole connection) stuck
		// forever with nothing reporting it (#5); log once, keep waiting either way
		tonHostNameStuck(IN := TRUE, PT := T#30S);
		IF tonHostNameStuck.Q AND NOT bHostNameStuckLogged THEN
			bHostNameStuckLogged := TRUE;
			ADSLOGSTR(ADSLOG_MSGTYPE_ERROR OR ADSLOG_MSGTYPE_LOG, 'MQTT: FB_GetHostName has not returned a hostname after 30s, still waiting', '');
		END_IF
	END_IF
	
1:
	// set parameters
    fbMqttClient.sHostName      := sHostName;
    fbMqttClient.nHostPort      := nHostPort;
    fbMqttClient.sClientId      := HostName;
    fbMqttClient.sTopicPrefix   := '';
	fbMqttClient.nKeepAlive     := nKeepAlive;
    fbMqttClient.ipMessageQueue := fbMessageQueue;

	// last will: the broker publishes this (retained) if this client disconnects uncleanly
	// (crash, power loss, network loss), so a consumer can tell the PLC is actually gone instead
	// of telemetry just having gone quiet (#5). Paired with the explicit 'online' publish below
	// once actually connected, so the retained value on this topic always reflects current status
	sStatusTopic := CONCAT(sTopicPublish, '/status');
	sOfflinePayload := 'offline';
	fbMqttClient.stWill.sTopic := sStatusTopic;
	fbMqttClient.stWill.eQoS := TcIotMqttQos.AtLeastOnceDelivery;
	fbMqttClient.stWill.bRetain := TRUE;
	fbMqttClient.stWill.pPayload := ADR(sOfflinePayload);
	fbMqttClient.stWill.nPayloadSize := LEN2(ADR(sOfflinePayload));

	// connect
	fbMqttClient.Execute(bConnect := TRUE);
	IF fbMqttClient.bConnected THEN
		state := 2;
	END_IF

2:
  	// subscribe
	fbMqttClient.Execute(bConnect := TRUE);
	// QoS 1 so that a command (stop!) is not lost silently (#27). It only takes effect if the sender publishes
	// with QoS 1 too (the broker delivers at the lower of the two). A command can then arrive twice: a repeated
	// single-field track/slew finds the coordinate buffer consumed and is dropped, a repeated multi-field one goes
	// to the same target again; the other commands only set a state that is already set.
	IF fbMqttClient.Subscribe(sTopic:=sTopicSub, eQoS:=TcIotMqttQos.AtLeastOnceDelivery) THEN
		bConnected := TRUE;
		// birth message: overwrites the retained 'offline' left by an earlier unclean disconnect
		sOnlinePayload := 'online';
		fbMqttClient.Publish(sTopic := sStatusTopic, pPayload := ADR(sOnlinePayload), nPayloadSize := LEN2(ADR(sOnlinePayload)),
			eQoS := TcIotMqttQos.AtLeastOnceDelivery, bRetain := TRUE, bQueue := TRUE);
		state := 3;
	END_IF
	
3:
	// keep bConnected honest: reflect the live underlying client state
	bConnected := fbMqttClient.bConnected;
	
	// if the broker dropped us, fall back to reconnect
	IF NOT fbMqttClient.bConnected THEN
		bConnected := FALSE;
		state := 1;
	END_IF
	
	// receive queued messages
	fbMqttClient.Execute(bConnect := TRUE);
	IF fbMessageQueue.nQueuedMessages > 0 THEN
		IF fbMessageQueue.Dequeue(fbMessage:=fbMessage) THEN
			fbMessage.GetTopic(pTopic:=ADR(sTopicRcv), nTopicSize:=SIZEOF(sTopicRcv) );
			fbMessage.GetPayload(pPayload:=ADR(sPayloadRcv), nPayloadSize:=SIZEOF(sPayloadRcv), bSetNullTermination:=TRUE);
			ADSLOGSTR(ADSLOG_MSGTYPE_HINT OR ADSLOG_MSGTYPE_LOG, 'MQTT %s', sPayloadRcv);
			IF sTopicRcv = sTopicSub THEN
				_handleMQTTMessage(sPayloadRcv);
			END_IF // measurement
		END_IF // Topic
		sPayloadRcv := '';
    END_IF // Dequeue
	
END_CASE

METHOD ABSTRACT _handleMQTTMessage : BOOL
VAR_INPUT
	sPayloadRcv	: STRING(255);
END_VAR
END_METHOD

METHOD Publish : BOOL
VAR_INPUT
	domain			: STRING(255) := 'environment';
	location		: STRING(255) := 'roof';
	parameter		: STRING(255);
	value			: STRING(255);
END_VAR
VAR_OUTPUT
	published	: BOOL;
END_VAR
END_METHOD

METHOD PublishLog : BOOL
VAR_INPUT
	level		: STRING(255) := 'INFO';
	message		: STRING(255);
END_VAR
VAR_OUTPUT
	published	: BOOL;
END_VAR
END_METHOD

END_FUNCTION_BLOCK

// ---- POUs/Comm/FB_Comm_MQTT_Influx.TcPOU
FUNCTION_BLOCK FB_Comm_MQTT_Influx EXTENDS FB_Comm_MQTT
VAR_INPUT
END_VAR
VAR_OUTPUT
END_VAR
VAR
	RaDec		: ST_RaDecCoordinate := (RightAscension := GVL_Math.LREAL_MIN, Declination := GVL_Math.LREAL_MIN);
	AltAz		: ST_AltAzCoordinate := (Altitude := GVL_Math.LREAL_MIN, Azimuth := GVL_Math.LREAL_MIN);
	dropped		: INT := 0;	// lines too long for the 255 character buffer, not published
	deliveryFailed	: INT := 0;	// fbMqttClient.Publish() returned FALSE (e.g. client busy/not connected); periodic telemetry, not retried on purpose (#5)
	// 0.0 doubles as "no data received yet" and FB_CO_REFRACT's own "estimate from altitude"
	// sentinel, so a consumer can pass these straight through with no guard needed.
	Temperature	: LREAL := 0.0;	// last received ambient temperature (deg C), set via MQTT by an external weather-station bridge
	Humidity	: LREAL := GVL_Math.LREAL_MIN;	// last received relative humidity (%); unconsumed anywhere today
	Pressure	: LREAL := 0.0;	// last received atmospheric pressure (hPa)

	// revert Temperature/Pressure to their safe defaults if nothing fresh arrives for a while,
	// instead of serving an arbitrarily stale weather reading forever
	bWeatherMessageReceived	: BOOL;
	tonWeatherStale			: TON := (PT := T#10M);
END_VAR

SUPER^();

tonWeatherStale(IN := NOT bWeatherMessageReceived, PT := T#10M);
bWeatherMessageReceived := FALSE;
IF tonWeatherStale.Q THEN
	Temperature := 0.0;
	Pressure := 0.0;
END_IF

METHOD _handleMQTTMessage : BOOL
VAR_INPUT
	sPayloadRcv		: STRING(255);
END_VAR
// A message can carry several parameter=value pairs (command a=1,b=2). Data fields (rightascension, declination,
// elevation, azimuth, ...) are applied first and track/slew last, so they always use the coordinates of this
// message, whatever the field order; for a single-field message nothing changes (BROTLib#39).
_DispatchPass(sPayloadRcv := sPayloadRcv, bVerbPass := FALSE);
_DispatchPass(sPayloadRcv := sPayloadRcv, bVerbPass := TRUE);
END_METHOD

// Runs one parameter=value pair of a 'command' message. Same dispatch as before the multi-field change (BROTLib#39).
METHOD PRIVATE _ApplyField
VAR_INPUT
	parameter		: STRING(255);
	value			: STRING(255);
	sPayloadRcv		: STRING(255);	// the whole payload, only for the log messages
END_VAR
VAR
	fValue			: LREAL;	// a number accepted by _ParseLREAL, before it is written
END_VAR
IF parameter = 'power' AND Telescope <> 0 THEN
	// there is no power-off command: Park() serves that role
	IF STRING_TO_UINT(value) = 1 THEN
		Telescope.CoverAutoOpen := TRUE;
		Telescope.Init();
	ELSIF STRING_TO_UINT(value) = 2 THEN
		Telescope.CoverAutoOpen := FALSE;
		Telescope.Init();
	ELSE
		ADSLOGSTR( ADSLOG_MSGTYPE_WARN OR ADSLOG_MSGTYPE_LOG, 'MQTT power: unrecognized value (want 1 or 2) %s', sPayloadRcv);
	END_IF
ELSIF parameter = 'park' AND Telescope <> 0 THEN
	Telescope.Park();
ELSIF parameter = 'gohome' AND Telescope <> 0 THEN
	Telescope.Home();
ELSIF parameter = 'track' AND Telescope <> 0 THEN
	// rightascension/declination are buffered here: they arrive either as separate messages beforehand (pyBROT,
	// BROTgui today) or in the same message as track (the data pass in _DispatchPass runs first, BROTLib#39);
	// an incomplete pair is dropped with a log entry
	IF RaDec.RightAscension > GVL_Math.LREAL_MIN AND RaDec.Declination > GVL_Math.LREAL_MIN THEN
		Telescope.Track(RaDec.RightAscension, RaDec.Declination);
	ELSE
		ADSLOGSTR( ADSLOG_MSGTYPE_WARN OR ADSLOG_MSGTYPE_LOG, 'MQTT track: rightascension/declination incomplete, command dropped %s', sPayloadRcv);
	END_IF
	RaDec.RightAscension := GVL_Math.LREAL_MIN;
	RaDec.Declination := GVL_Math.LREAL_MIN;
ELSIF parameter = 'slew' AND Telescope <> 0 THEN
	// see 'track' above -- same buffer-and-consume pattern, same incomplete-pair gap
	IF AltAz.Azimuth > GVL_Math.LREAL_MIN AND AltAz.Altitude > GVL_Math.LREAL_MIN THEN
		Telescope.Slew(AltAz.Azimuth, AltAz.Altitude);
	ELSE
		ADSLOGSTR( ADSLOG_MSGTYPE_WARN OR ADSLOG_MSGTYPE_LOG, 'MQTT slew: azimuth/elevation incomplete, command dropped %s', sPayloadRcv);
	END_IF
	AltAz.Azimuth := GVL_Math.LREAL_MIN;
	AltAz.Altitude := GVL_Math.LREAL_MIN;
ELSIF parameter = 'stop' AND Telescope <> 0 THEN
	Telescope.Stop();
ELSIF parameter = 'reset' AND Telescope <> 0 THEN
	Telescope.Reset();
ELSIF parameter = 'nasmyth' AND Nasmyth <> 0 THEN
	IF _ParseLREAL(parameter := parameter, value := value, fMin := 0.0, fMax := 255.0, fValue => fValue) THEN
		Nasmyth.SetNasmyth(LREAL_TO_USINT(fValue));
	END_IF
// Every number below goes through _ParseLREAL: text that is not a number, NaN/inf and values outside the range
// are rejected with a log entry instead of being written (#27). The ranges only catch garbage; the limits of the
// mount, focus and derotator are still the consumer's job. Angles in degrees.
// A rejected coordinate clears its buffer, so a following track/slew is dropped as incomplete instead of using
// a value buffered by an earlier message.
ELSIF parameter = 'rightascension' THEN
	IF NOT _ParseLREAL(parameter := parameter, value := value, fMin := 0.0, fMax := 360.0, fValue => RaDec.RightAscension) THEN
		RaDec.RightAscension := GVL_Math.LREAL_MIN;
	END_IF
ELSIF parameter = 'declination' THEN
	IF NOT _ParseLREAL(parameter := parameter, value := value, fMin := -90.0, fMax := 90.0, fValue => RaDec.Declination) THEN
		RaDec.Declination := GVL_Math.LREAL_MIN;
	END_IF
ELSIF parameter = 'elevation' THEN
	IF NOT _ParseLREAL(parameter := parameter, value := value, fMin := -90.0, fMax := 90.0, fValue => AltAz.Altitude) THEN
		AltAz.Altitude := GVL_Math.LREAL_MIN;
	END_IF
ELSIF parameter = 'azimuth' THEN
	IF NOT _ParseLREAL(parameter := parameter, value := value, fMin := -360.0, fMax := 360.0, fValue => AltAz.Azimuth) THEN
		AltAz.Azimuth := GVL_Math.LREAL_MIN;
	END_IF
ELSIF parameter = 'temperature' THEN
	// deg C; 0.0 is also the "no data" sentinel, see the declaration
	IF _ParseLREAL(parameter := parameter, value := value, fMin := -60.0, fMax := 60.0, fValue => fValue) THEN
		Temperature := fValue;
		bWeatherMessageReceived := TRUE;
	END_IF
ELSIF parameter = 'humidity' THEN
	IF _ParseLREAL(parameter := parameter, value := value, fMin := 0.0, fMax := 100.0, fValue => fValue) THEN
		Humidity := fValue;
		bWeatherMessageReceived := TRUE;
	END_IF
ELSIF parameter = 'pressure' THEN
	// hPa; 0.0 is FB_CO_REFRACT's "estimate from altitude" sentinel and stays allowed
	IF _ParseLREAL(parameter := parameter, value := value, fMin := 0.0, fMax := 1100.0, fValue => fValue) THEN
		Pressure := fValue;
		bWeatherMessageReceived := TRUE;
	END_IF
ELSIF parameter = 'dut1' AND AltAzTelescope <> 0 THEN
	// seconds; |UT1-UTC| is kept below 0.9 s by definition
	IF _ParseLREAL(parameter := parameter, value := value, fMin := -1.0, fMax := 1.0, fValue => fValue) THEN
		AltAzTelescope.Dut1 := fValue;
	END_IF
ELSIF parameter = 'focus' AND Focus <> 0 THEN
	// unit and travel depend on the telescope; this only rejects garbage, the focus axis enforces its limits
	IF _ParseLREAL(parameter := parameter, value := value, fMin := -1.0E6, fMax := 1.0E6, fValue => fValue) THEN
		Focus.Position := fValue;
	END_IF
ELSIF parameter = 'cover_open' AND MirrorCovers <> 0 THEN
	MirrorCovers.Open();
ELSIF parameter = 'cover_close' AND MirrorCovers <> 0 THEN
	MirrorCovers.Close();	
ELSIF parameter = 'dome_open' THEN
	IF Dome <> 0 THEN
		Dome.Open();
	ELSIF Roof <> 0 THEN
		Roof.Open();
	END_IF
ELSIF parameter = 'dome_close' THEN
	IF Dome <> 0 THEN
		Dome.Close();
	ELSIF Roof <> 0 THEN
		Roof.Close();
	END_IF
ELSIF parameter = 'dome_stop' AND (Dome <> 0 OR Roof <> 0) THEN
	IF Dome <> 0 THEN
		Dome.Stop();
	ELSIF Roof <> 0 THEN
		Roof.Stop();
	END_IF		
ELSIF parameter = 'dome_park' AND Dome <> 0 THEN
	Dome.Park();
ELSIF parameter = 'dome_track' AND Dome <> 0 THEN
	IF value = '1'THEN
		Dome.Track();
	ELSE
		Dome.StopTrack();
	END_IF	
ELSIF parameter = 'dome_reset' AND Dome <> 0 THEN
	Dome.Reset();
ELSIF parameter = 'filter' AND Filter <> 0 THEN
	// garbage used to become filter 0
	IF _ParseLREAL(parameter := parameter, value := value, fMin := 0.0, fMax := 255.0, fValue => fValue) THEN
		Filter.SetFilter(LREAL_TO_USINT(fValue));
	END_IF
ELSIF (parameter = 'derotator' OR parameter = 'derotatoroffset') AND AltAzTelescope <> 0 THEN
	// two client-facing names for the same thing -- I_AltAzTelescope only has one derotator
	// property (DerotatorOffset), there's no separate "absolute derotator position" concept
	IF _ParseLREAL(parameter := parameter, value := value, fMin := -360.0, fMax := 360.0, fValue => fValue) THEN
		AltAzTelescope.DerotatorOffset := fValue;
	END_IF
// pointing offsets: 10 degrees is far beyond any real offset. Near the zenith the consumers still divide the
// azimuth offset by COS(elevation), so they need their own cap there (#27).
ELSIF parameter = 'elevationoffset' AND AltAzTelescope <> 0 THEN
	IF _ParseLREAL(parameter := parameter, value := value, fMin := -10.0, fMax := 10.0, fValue => fValue) THEN
		AltAzTelescope.AltitudeOffset := fValue;
	END_IF
ELSIF parameter = 'azimuthoffset' AND AltAzTelescope <> 0 THEN
	IF _ParseLREAL(parameter := parameter, value := value, fMin := -10.0, fMax := 10.0, fValue => fValue) THEN
		AltAzTelescope.AzimuthOffset := fValue;
	END_IF
ELSIF parameter = 'declinationoffset' AND RaDecTelescope <> 0 THEN
	IF _ParseLREAL(parameter := parameter, value := value, fMin := -10.0, fMax := 10.0, fValue => fValue) THEN
		RaDecTelescope.DeclinationOffset := fValue;
	END_IF
ELSIF parameter = 'hourangleoffset' AND RaDecTelescope <> 0 THEN
	IF _ParseLREAL(parameter := parameter, value := value, fMin := -10.0, fMax := 10.0, fValue => fValue) THEN
		RaDecTelescope.HourAngleOffset := fValue;
	END_IF
ELSE
	ADSLOGSTR( ADSLOG_MSGTYPE_WARN OR ADSLOG_MSGTYPE_LOG, 'MQTT not understood %s', sPayloadRcv);
END_IF
END_METHOD

// Converts the value of a command field to a number. Returns FALSE, with a log entry, when the text is not a
// number (STRING_TO_LREAL would turn it into 0.0, a valid coordinate), or when the number is NaN, infinite or
// outside fMin..fMax (#27). fValue is only meaningful when it returns TRUE.
METHOD PRIVATE _ParseLREAL : BOOL
VAR_INPUT
	parameter		: STRING(255);
	value			: STRING(255);
	fMin			: LREAL;
	fMax			: LREAL;
END_VAR
VAR_OUTPUT
	fValue			: LREAL;
END_VAR
fValue := 0.0;
IF F_IsNumericValue(sValue := value) THEN
	fValue := STRING_TO_LREAL(value);
	// written this way round so that NaN, which fails every comparison, is rejected too
	_ParseLREAL := fValue >= fMin AND fValue <= fMax;
END_IF
IF NOT _ParseLREAL THEN
	ADSLOGSTR( ADSLOG_MSGTYPE_WARN OR ADSLOG_MSGTYPE_LOG, 'MQTT %s rejected: not a number or out of range',
		CONCAT(CONCAT(parameter, '='), value));
END_IF
END_METHOD

// Walks the parameter=value pairs of a payload via FB_InfluxMessage.remaining and applies the ones that belong to
// this pass: bVerbPass FALSE applies everything except track/slew, TRUE applies only track/slew. Running the
// data pass first means track/slew always see the coordinates of the SAME message (any field order), and a
// single-field message behaves exactly as before. At most MAX_FIELDS pairs are walked per message.
METHOD PRIVATE _DispatchPass
VAR_INPUT
	sPayloadRcv		: STRING(255);
	bVerbPass		: BOOL;
END_VAR
VAR
	influxMessage	: FB_InfluxMessage;
	sNext			: STRING(255);
	nFields			: INT;
	bVerb			: BOOL;
END_VAR
VAR CONSTANT
	MAX_FIELDS		: INT := 8;
END_VAR
sNext := sPayloadRcv;
WHILE sNext <> '' AND nFields < MAX_FIELDS DO
	nFields := nFields + 1;
	influxMessage(sPayload := sNext);
	IF influxMessage.measurement <> 'command' THEN
		RETURN;
	END_IF
	bVerb := influxMessage.parameter = 'track' OR influxMessage.parameter = 'slew';
	IF bVerb = bVerbPass THEN
		_ApplyField(parameter := influxMessage.parameter, value := influxMessage.value, sPayloadRcv := sPayloadRcv);
	END_IF
	sNext := influxMessage.remaining;
END_WHILE
IF sNext <> '' AND NOT bVerbPass THEN
	ADSLOGSTR( ADSLOG_MSGTYPE_WARN OR ADSLOG_MSGTYPE_LOG, 'MQTT more than 8 fields in one message, the rest is ignored %s', sPayloadRcv);
END_IF
END_METHOD

METHOD Publish : BOOL
VAR_INPUT
	domain			: STRING(255) := 'environment';
	location		: STRING(255) := 'roof';
	parameter		: STRING(255);
	value			: STRING(255);
END_VAR
VAR_OUTPUT
	published	: BOOL;
END_VAR
VAR
	sPayloadPub		: STRING(255) := '';
	fbFormat		: FB_FormatString;
	bError			: BOOL;
	nErrID			: UDINT;
	retain_message	: BOOL := FALSE;
	bIsBool			: BOOL;
	sDomain			: STRING(255);
	sLocation		: STRING(255);
	sHost			: STRING(255);
	sKey			: STRING(255);
	sFieldVal		: STRING(255);
	sTopic			: STRING(255);
	sTimestamp		: STRING(255);	// F_STRING takes a T_MaxString by reference
	sFormat			: STRING(40);
END_VAR
//sPayloadPub := 'environment,location=roof,host=CX-4E6032 ';
// tag values and the field key are escaped (a space or comma in the host name would break the line); the field
// value is typed by F_InfluxFieldValue: integer 'i', float, boolean or quoted string
sDomain := F_EscapeInfluxTag(domain, FALSE);
sLocation := F_EscapeInfluxTag(location, TRUE);
sHost := F_EscapeInfluxTag(HostName, TRUE);
sKey := F_EscapeInfluxTag(parameter, TRUE);
sFieldVal := F_InfluxFieldValue(value);

// retain message if value is boolean: booleans are meant to be published on change only, so a subscriber that
// connects later gets the current state from the broker
bIsBool := (value = 'TRUE') OR (value = 'FALSE') OR (value = 'true') OR (value = 'false');
retain_message := bIsBool;

// a retained line carries the time it was published, so a replay after a Telegraf restart is stored at that time
// and not at the time of the replay (#38). Consumers must accept the optional timestamp (pyBROT#40).
sTimestamp := '';
IF retain_message THEN
	sTimestamp := F_InfluxTimestamp(F_GetSystemTime());
END_IF
IF sTimestamp <> '' THEN
	sFormat := '%s,location=%s,host=%s %s=%s %s';
ELSE
	sFormat := '%s,location=%s,host=%s %s=%s';
END_IF

fbFormat(
	sFormat 	:= sFormat,
	arg1 		:= F_STRING(sDomain),
	arg2 		:= F_STRING(sLocation),
	arg3 		:= F_STRING(sHost),
	arg4 		:= F_STRING(sKey),
	arg5 		:= F_STRING(sFieldVal),
	arg6 		:= F_STRING(sTimestamp),
	sOut 		=> sPayloadPub,
	bError 		=> bError,
	nErrID 		=> nErrID
);

// a line that did not fit the buffer is cut off and would be invalid (or wrong): do not publish it
IF bError OR LEN(sPayloadPub) >= 255 THEN
	published := FALSE;
	IF dropped < 32767 THEN
		dropped := dropped + 1;
	END_IF
	IF dropped = 1 OR (dropped MOD 100) = 0 THEN
		ADSLOGSTR(ADSLOG_MSGTYPE_WARN OR ADSLOG_MSGTYPE_LOG, 'Influx line too long, not published: %s', parameter);
	END_IF
	Publish := published;
	RETURN;
END_IF

// publish under a per-subsystem sub-topic (domain is already the Influx measurement, e.g.
// 'telescope'/'power'/'electronics'/'hydraulics'/'diagnostics') so a consumer that only cares
// about one subsystem can subscribe to just that sub-topic instead of the whole site's firehose
sTopic := CONCAT(CONCAT(sTopicPublish, '/'), domain);

// bQueue left FALSE on purpose: this is periodic telemetry (republished every 1-5s or on the
// static-fields timer), so a dropped publish under load is self-healing next cycle -- queuing
// would just build a backlog of stale values behind whatever caused the client to be busy.
// One-time events (PublishLog) get bQueue := TRUE instead, see there. (#5)
published := fbMqttClient.Publish(
	sTopic			:= sTopic,
	pPayload		:= ADR(sPayloadPub),
	nPayloadSize	:= LEN2(ADR(sPayloadPub)),
	eQoS			:= TcIotMqttQos.AtMostOnceDelivery,
	bRetain			:= retain_message,
	bQueue			:= FALSE
);

IF NOT published THEN
	IF deliveryFailed < 32767 THEN
		deliveryFailed := deliveryFailed + 1;
	END_IF
	IF deliveryFailed = 1 OR (deliveryFailed MOD 100) = 0 THEN
		ADSLOGSTR(ADSLOG_MSGTYPE_WARN OR ADSLOG_MSGTYPE_LOG, 'MQTT publish failed (client busy/not connected): %s', parameter);
	END_IF
END_IF

Publish := published;
END_METHOD

METHOD PublishLog : BOOL
VAR_INPUT
	level		: STRING(255) := 'INFO';
	message		: STRING(255);
END_VAR
VAR
	sPayloadPub		: STRING(255) := '';
	fbFormat		: FB_FormatString;
	bError			: BOOL;
	nErrID			: UDINT;
	sEscapedMessage	: STRING(255);
	sHost			: STRING(255);
	sLevel			: STRING(255);
	nMaxMessage		: INT;
END_VAR
VAR_OUTPUT
	published	: BOOL;
END_VAR
//sPayloadPub := 'environment,location=roof,host=CX-4E6032 ';
sHost := F_EscapeInfluxTag(HostName, TRUE);
sLevel := F_EscapeInfluxTag(level, TRUE);
sEscapedMessage := F_EscapeInfluxString(message);

// a long message is shortened so that the line fits the 255 character buffer and its closing quote is kept:
// 255 minus 'log,host=' (9), ',level=' (7), ' message="' (10) and the closing '"' (1)
nMaxMessage := 255 - 27 - LEN(sHost) - LEN(sLevel);
sEscapedMessage := F_TruncateInfluxEscaped(sEscapedMessage, nMaxMessage);

fbFormat(
	sFormat := 'log,host=%s,level=%s message="%s"',
	arg1 	:= F_STRING(sHost),
	arg2 	:= F_STRING(sLevel),
	arg3 	:= F_STRING(sEscapedMessage),
	sOut 	=> sPayloadPub,
	bError 	=> bError,
	nErrID 	=> nErrID
);

// still too long (very long host name or level): publish nothing rather than a broken line
IF bError OR LEN(sPayloadPub) >= 255 THEN
	published := FALSE;
	PublishLog := published;
	RETURN;
END_IF

// bQueue TRUE: unlike Publish()'s periodic telemetry, a log/event message is one-time -- if the
// client can't send it immediately, queue it for retry instead of losing it silently (#5)
published := fbMqttClient.Publish(
	sTopic			:= sTopicLog,
	pPayload		:= ADR(sPayloadPub),
	nPayloadSize	:= LEN2(ADR(sPayloadPub)),
	eQoS			:= TcIotMqttQos.AtMostOnceDelivery,
	bRetain			:= FALSE,
	bQueue			:= TRUE
);

PublishLog := published;
END_METHOD

END_FUNCTION_BLOCK

// ---- POUs/Comm/F_IsNumericValue.TcPOU
FUNCTION F_IsNumericValue : BOOL
VAR_INPUT
	sValue		: STRING(255);
END_VAR
VAR
	i				: INT;
	nLen			: INT;
	bSeenDigit		: BOOL := FALSE;
	bSeenDot		: BOOL := FALSE;
	bSeenExp		: BOOL := FALSE;
	bSeenExpDigit	: BOOL := FALSE;
	bPrevWasExp		: BOOL := FALSE;
	c			: STRING(1);
END_VAR

F_IsNumericValue := FALSE;
nLen := LEN(sValue);
IF nLen = 0 THEN
	RETURN;
END_IF

FOR i := 1 TO nLen DO
	c := MID(sValue, 1, i);
	IF (c = '-' OR c = '+') AND (i = 1 OR bPrevWasExp) THEN
		; // leading sign, or sign right after 'e'/'E', OK
	ELSIF c = '.' AND NOT bSeenDot AND NOT bSeenExp THEN
		bSeenDot := TRUE;
	ELSIF (c = 'e' OR c = 'E') AND NOT bSeenExp AND bSeenDigit THEN
		bSeenExp := TRUE;
	ELSIF c >= '0' AND c <= '9' THEN
		IF bSeenExp THEN
			bSeenExpDigit := TRUE;
		ELSE
			bSeenDigit := TRUE;
		END_IF
	ELSE
		RETURN; // any other char -> not purely numeric
	END_IF
	bPrevWasExp := (c = 'e' OR c = 'E');
END_FOR

// a trailing exponent marker with no digits (e.g. "1e") is not a complete number
F_IsNumericValue := bSeenDigit AND (NOT bSeenExp OR bSeenExpDigit);

END_FUNCTION

// ---- POUs/FB_InfluxMessage.TcPOU
FUNCTION_BLOCK FB_InfluxMessage
VAR_INPUT
	// payload string received
	sPayload:	STRING(255);
END_VAR
VAR_OUTPUT
	// measurement string (first word)
	measurement:	STRING(255) := '';
	// parameter (variable name)
	parameter:		STRING(255) := '';
	// value (variable content)
	value:			STRING(255) := '';
	// the payload for the NEXT parameter=value pair ("measurement[,tags] rest-of-field-set[ timestamp]"),
	// '' if this was the last pair. Feed it back in as sPayload to walk a multi-field message.
	remaining:		STRING(255) := '';
END_VAR
VAR
	space_position:		INT;
	//equial_position:	INT;
	comma_position:		INT;
	measurement_tags:	STRING(255);
	parameter_value: 	STRING(255);
	bResultSplit: 		BOOL;
	sRest:				STRING(255);
	// definition of the space separator
	spaceSeparator:		STRING(1) := ' ';
	// definition of the comma separator
	commaSeparator:		STRING(1) := ',';
	// definition of the equial sign separator
	equialSeparator:	STRING(1) := '=';
END_VAR

(* 
parse message in influx format:
	measurement parameter=value
	measurement,tag1=tag1value parameter=value
	measurement,tag1=tag1value parameter1=value1,parameter2=value2 [timestamp]

Returns the FIRST parameter=value pair. If there are more, 'remaining' holds a complete payload for the next
pair (measurement and tags in front, timestamp kept at the end), so the caller feeds it straight back in.
Tags are accepted but not returned. A quoted string value that contains a comma or a space is not handled.
*)

// start from empty outputs every call: a caller that reuses the instance must not see the previous pair again
measurement := '';
parameter := '';
value := '';
remaining := '';

//separate measurement from parameter, value
bResultSplit := FindAndSplit( pSeparator     := ADR(spaceSeparator), pSrcString := ADR(sPayload), 
                              pLeftString    := ADR(measurement_tags), nLeftSize  := SIZEOF(measurement_tags), 
                              pRightString   := ADR(parameter_value), nRightSize := SIZEOF(parameter_value),
                              bSearchFromRight := FALSE );
IF NOT bResultSplit THEN
	RETURN;
END_IF
// look for tags attached to the measurement
comma_position := FIND(measurement_tags, commaSeparator);
IF comma_position = 0 THEN
	measurement := measurement_tags;
ELSE
	measurement := LEFT(measurement_tags, comma_position-1);
END_IF
// dissect the parameter=value part
comma_position := FIND(parameter_value, commaSeparator);
IF comma_position = 0 THEN
	// we have only one parameter value pair
	bResultSplit := FindAndSplit( pSeparator     := ADR(equialSeparator), pSrcString := ADR(parameter_value), 
                              pLeftString    := ADR(parameter), nLeftSize  := SIZEOF(parameter), 
                              pRightString   := ADR(value), nRightSize := SIZEOF(value),
                              bSearchFromRight := FALSE );

ELSE
	// we have more than one parameter value pair: everything after the first comma is the next pair(s),
	// handed back with the measurement and tags in front (the space between them was consumed above)
	sRest := MID(parameter_value, LEN(parameter_value) - comma_position, comma_position + 1);
	remaining := CONCAT(CONCAT(measurement_tags, spaceSeparator), sRest);
	parameter_value := LEFT(parameter_value, comma_position-1);
	bResultSplit := FindAndSplit( pSeparator     := ADR(equialSeparator), pSrcString := ADR(parameter_value), 
                              pLeftString    := ADR(parameter), nLeftSize  := SIZEOF(parameter), 
                              pRightString   := ADR(value), nRightSize := SIZEOF(value),
                              bSearchFromRight := FALSE );
END_IF

// a trailing Influx timestamp (measurement[,tags] field_set timestamp) ends up appended to value,
// since only the first space in the whole payload is split off above; drop it and anything after
// the first remaining space. A genuine quoted string value could itself contain a space, but this
// parser doesn't handle that either way (see the module comment's TODOs)
space_position := FIND(value, spaceSeparator);
IF space_position > 0 THEN
	value := LEFT(value, space_position-1);
END_IF

// strip the surrounding quotes Influx line protocol uses for a string-typed field value
IF LEN(value) >= 2 AND LEFT(value,1) = '"' AND RIGHT(value,1) = '"' THEN
	value := MID(value, LEN(value)-2, 2);
END_IF

END_FUNCTION_BLOCK

// ---- POUs/Comm/F_EscapeInfluxTag.TcPOU
// Escapes a tag value or a field key for InfluxDB line protocol: a comma, a space and (unless it is a measurement
// name, where '=' needs no escape) an equals sign get a leading backslash. Without it a space in e.g. the host
// name ends the tag set and breaks the line.
FUNCTION F_EscapeInfluxTag : STRING(255)
VAR_INPUT
	sValue			: STRING(255);
	bEscapeEquals	: BOOL;		// TRUE for tag values and field keys, FALSE for a measurement name
END_VAR
VAR
	i, nLen		: INT;
	c			: STRING(1);
	sOut		: STRING(255) := '';
END_VAR

nLen := LEN(sValue);
FOR i := 1 TO nLen DO
	c := MID(sValue, 1, i);
	IF c = ',' OR c = ' ' OR (c = '=' AND bEscapeEquals) THEN
		sOut := CONCAT(sOut, CONCAT('\', c));
	ELSE
		sOut := CONCAT(sOut, c);
	END_IF
END_FOR

F_EscapeInfluxTag := sOut;

END_FUNCTION

// ---- POUs/Comm/F_InfluxFieldValue.TcPOU
// Field value as it is written in an InfluxDB line protocol line, decided from the text of the value:
//   integer (no '.', no exponent)  -> trailing 'i'       15    -> 15i
//   number with '.' or exponent    -> float, as is        15.5  -> 15.5,  1e5 -> 1e5
//   TRUE / FALSE / true / false    -> boolean, as is
//   anything else                  -> quoted, with " and \ escaped
// Note that the same field flips between integer and float if its text flips between '15' and '15.5' (see
// F_IsNumericValue); only a typed publisher would fix that.
FUNCTION F_InfluxFieldValue : STRING(255)
VAR_INPUT
	sValue		: STRING(255);
END_VAR
VAR
	bIsBool		: BOOL;
	bIsNumeric	: BOOL;
	bIsInteger	: BOOL;
END_VAR

bIsBool := (sValue = 'TRUE') OR (sValue = 'FALSE') OR (sValue = 'true') OR (sValue = 'false');
bIsNumeric := F_IsNumericValue(sValue);
// 1e5 has no '.', but appending 'i' to it is invalid line protocol: a number with an exponent is a float
bIsInteger := bIsNumeric AND (FIND(sValue, '.') = 0) AND (FIND(sValue, 'e') = 0) AND (FIND(sValue, 'E') = 0);

IF bIsInteger THEN
	F_InfluxFieldValue := CONCAT(sValue, 'i');
ELSIF bIsBool OR bIsNumeric THEN
	F_InfluxFieldValue := sValue;
ELSE
	F_InfluxFieldValue := CONCAT('"', CONCAT(F_EscapeInfluxString(sValue), '"'));
END_IF

END_FUNCTION

// ---- POUs/Comm/F_EscapeInfluxString.TcPOU
FUNCTION F_EscapeInfluxString : STRING(255)
VAR_INPUT
	sValue		: STRING(255);
END_VAR
VAR
	i, nLen		: INT;
	c			: STRING(1);
	sOut		: STRING(255) := '';
END_VAR

nLen := LEN(sValue);
FOR i := 1 TO nLen DO
	c := MID(sValue, 1, i);
	IF c = '"' OR c = '\' THEN
		sOut := CONCAT(sOut, CONCAT('\', c));
	ELSE
		sOut := CONCAT(sOut, c);
	END_IF
END_FOR

F_EscapeInfluxString := sOut;

END_FUNCTION

// ---- POUs/Comm/F_InfluxTimestamp.TcPOU
// Influx line-protocol timestamp (unix nanoseconds) from a Windows FILETIME (100 ns since 1601-01-01 UTC, as
// returned by F_GetSystemTime). Empty for a time before 1970, so the caller leaves the timestamp off and the
// receiver stamps the line instead. (#38)
FUNCTION F_InfluxTimestamp : STRING(20)
VAR_INPUT
	nFileTime	: ULINT;
END_VAR
VAR CONSTANT
	FILETIME_UNIX_EPOCH	: ULINT := 116444736000000000;	// 1970-01-01 00:00:00 UTC as FILETIME
END_VAR

IF nFileTime < FILETIME_UNIX_EPOCH THEN
	F_InfluxTimestamp := '';
	RETURN;
END_IF

F_InfluxTimestamp := ULINT_TO_STRING((nFileTime - FILETIME_UNIX_EPOCH) * 100);

END_FUNCTION

// ---- POUs/Comm/F_TruncateInfluxEscaped.TcPOU
// Shortens an already escaped string to at most nMaxLen characters without cutting an escape pair in half. A cut
// that leaves a lone backslash at the end would escape the closing quote of a quoted string field.
FUNCTION F_TruncateInfluxEscaped : STRING(255)
VAR_INPUT
	sEscaped	: STRING(255);
	nMaxLen		: INT;
END_VAR
VAR
	sOut			: STRING(255);
	i, nBackslashes	: INT;
END_VAR

IF nMaxLen < 0 THEN
	nMaxLen := 0;
END_IF
IF LEN(sEscaped) <= nMaxLen THEN
	F_TruncateInfluxEscaped := sEscaped;
	RETURN;
END_IF

sOut := LEFT(sEscaped, nMaxLen);
// an odd number of backslashes at the end means the cut is between a backslash and the character it escapes
nBackslashes := 0;
i := LEN(sOut);
WHILE i > 0 AND MID(sOut, 1, i) = '\' DO
	nBackslashes := nBackslashes + 1;
	i := i - 1;
END_WHILE
IF (nBackslashes MOD 2) = 1 THEN
	sOut := LEFT(sOut, LEN(sOut) - 1);
END_IF

F_TruncateInfluxEscaped := sOut;

END_FUNCTION

// ---- POUs/Debug/FB_InfoConnection.TcPOU
// Decodes the Map State / Map Diag bytes of a TwinSAFE (FSoE) connection into text for debugging.
// Map Diag (Beckhoff H0003 "TwinSAFE Diagnostik"): bits 0-3 hold a numeric error code (1..12),
// bits 4-7 are independent flags. Bit 4 is confirmed there; the texts of bits 5-7 are the ones this
// block always used.
FUNCTION_BLOCK FB_InfoConnection
VAR_INPUT
	stInfoData	:ST_InfoDataConnection;
END_VAR
VAR_OUTPUT
	sState		:STRING;
	sDiag		:STRING(255);	// error code text followed by any set flags, separated by '; '
	nDiagCode	:USINT;			// bits 0-3 of usiMapDiag
	bSlaveError			:BOOL;	// bit 4: error detected by the FSoE slave
	bSlaveFailsafe		:BOOL;	// bit 5: FSoE slave reports failsafe value active
	bStartUp			:BOOL;	// bit 6: start-up
	bMasterFailsafe		:BOOL;	// bit 7: FSoE master reports failsafe value active
	bChannel1	:BOOL;
	bChannel2	:BOOL;
	bChannel3	:BOOL;
	bChannel4	:BOOL;
END_VAR

CASE stInfoData.usiMapState OF
	100: sState := 'State Reset';
	101: sState := 'State Session';
	102: sState := 'State Connection';
	103: sState := 'State Parameter';
	104: sState := 'State Data';
	105: sState := 'State Shutdown';
ELSE
	sState := 'Error';
END_CASE

// the low nibble is a number, not a set of bits: 3 is "Invalid Connection ID", not "Invalid Command"
nDiagCode := stInfoData.usiMapDiag AND 16#0F;
CASE nDiagCode OF
	0:  sDiag := '';
	1:  sDiag := 'Invalid Command';
	2:  sDiag := 'Unknown Command';
	3:  sDiag := 'Invalid Connection ID';
	4:  sDiag := 'Invalid CRC';
	5:  sDiag := 'Watchdog expired';
	6:  sDiag := 'Invalid FSoE address';
	7:  sDiag := 'Invalid data';
	8:  sDiag := 'Invalid Com.-Parameter length';
	9:  sDiag := 'Invalid Com.-Parameter';
	10: sDiag := 'Invalid User-Parameter length';
	11: sDiag := 'Invalid User-Parameter';
	12: sDiag := 'FSoE Master Reset';
ELSE
	sDiag := CONCAT('Unknown error code ', USINT_TO_STRING(nDiagCode));
END_CASE

// the high nibble is flags that can be set together with any code
bSlaveError		:= stInfoData.usiMapDiag.4;
bSlaveFailsafe	:= stInfoData.usiMapDiag.5;
bStartUp		:= stInfoData.usiMapDiag.6;
bMasterFailsafe	:= stInfoData.usiMapDiag.7;
IF bSlaveError THEN
	_Append('Error by FSoE Slave detected');
END_IF
IF bSlaveFailsafe THEN
	_Append('FSoE Slave reports Failsafe value active');
END_IF
IF bStartUp THEN
	_Append('StartUp');
END_IF
IF bMasterFailsafe THEN
	_Append('FSoE Master reports Failsafe value active');
END_IF
IF sDiag = '' THEN
	sDiag := 'No error';
END_IF

(*Signals*)
bChannel1 := stInfoData.bySignal.0;
bChannel2 := stInfoData.bySignal.1;
bChannel3 := stInfoData.bySignal.2;
bChannel4 := stInfoData.bySignal.3;

// Appends sText to sDiag, separated by '; ' when sDiag is not empty.
METHOD PRIVATE _Append
VAR_INPUT
	sText	: STRING;
END_VAR
IF sDiag <> '' THEN
	sDiag := CONCAT(sDiag, '; ');
END_IF
sDiag := CONCAT(sDiag, sText);
END_METHOD

END_FUNCTION_BLOCK

// ---- POUs/Debug/FB_InfoEStop.TcPOU
FUNCTION_BLOCK FB_InfoEStop
VAR_INPUT
	stInfoData		:ST_InfoDataFB;
END_VAR
VAR_OUTPUT
	sState			:STRING;
	sDiag			:STRING;
END_VAR

IF stInfoData.usiMapState= 0 THEN
	sState:='undefined';
ELSIF stInfoData.usiMapState= 1 THEN
	sState:='RUN';
ELSIF stInfoData.usiMapState= 2 THEN
	sState:='STOP';
ELSIF stInfoData.usiMapState= 3 THEN
	sState:='SAFE';
ELSIF stInfoData.usiMapState= 4 THEN
	sState:='ERROR';
ELSIF stInfoData.usiMapState= 5 THEN
	sState:='RESET';
ELSIF stInfoData.usiMapState= 6 THEN
	sState:='START';
ELSIF stInfoData.usiMapState= 8 THEN
	sState:='DELAYOUT';
ELSE
	sState:='Unknown';
END_IF

IF stInfoData.uiMapDiag = 0 THEN
	sDiag:='No error';
ELSIF stInfoData.uiMapDiag.0 THEN
	sDiag:='Discrepancy error input group 1';
ELSIF stInfoData.uiMapDiag.1 THEN
	sDiag:='Discrepancy error input group 2';
ELSIF stInfoData.uiMapDiag.2 THEN
	sDiag:='Discrepancy error input group 3';
ELSIF stInfoData.uiMapDiag.3 THEN
	sDiag:='Discrepancy error input group 4';
ELSIF stInfoData.uiMapDiag.4 THEN
	sDiag:='EDM Error EDM 1';
ELSIF stInfoData.uiMapDiag.5 THEN
	sDiag:='EDM Error EDM 2';
ELSE
	sDiag:='Unknown';
END_IF

END_FUNCTION_BLOCK

// ---- POUs/Debug/FB_InfoGroup.TcPOU
FUNCTION_BLOCK FB_InfoGroup
VAR_INPUT
	stInfoData	:ST_InfoDataGroup;
END_VAR
VAR_OUTPUT
	sState		:STRING;
END_VAR
VAR
END_VAR

IF stInfoData.usiMapState= 1 THEN
	sState:='RUN';
ELSIF stInfoData.usiMapState= 2 THEN
	sState:='STOP';
ELSIF stInfoData.usiMapState= 3 THEN
	sState:='SAFE';
ELSIF stInfoData.usiMapState= 4 THEN
	sState:='ERROR';
ELSIF stInfoData.usiMapState= 5 THEN
	sState:='RESET';
ELSE
	sState:='Unknown';
END_IF

END_FUNCTION_BLOCK

// ---- POUs/F_SetpointEnableExecute.TcPOU
// Next value of FB_Axis's MC_ExtSetPointGenEnable.Execute (#9). Pure logic, so it can be tested without an NC axis.
// After an error Execute drops: an MC block clears Error only when Execute falls, and only a later rising edge can
// enable it again (before #9 Execute stayed TRUE, so the axis could never track again). Failed then holds off a
// retry until Reset or the end of the track request, instead of retrying every second cycle.
FUNCTION F_SetpointEnableExecute : BOOL
VAR_INPUT
	Request		: BOOL;		// tracking wanted and possible (Tracking AND Ready AND Calibrated AND NOT StopAxis)
	Tracking	: BOOL;		// the track request itself; its end re-arms after an error
	Reset		: BOOL;		// FB_Axis.Reset; re-arms after an error
	Execute		: BOOL;		// the current Execute
	Busy		: BOOL;		// MC_ExtSetPointGenEnable outputs of the last call
	Done		: BOOL;
	Error		: BOOL;
END_VAR
VAR_IN_OUT
	Failed		: BOOL;		// TRUE from an error until Reset or the end of the track request
END_VAR

IF Error THEN
	Failed := TRUE;
	F_SetpointEnableExecute := FALSE;
	RETURN;
END_IF

IF Reset OR NOT Tracking THEN
	Failed := FALSE;
END_IF

IF Request AND NOT Failed THEN
	F_SetpointEnableExecute := TRUE;
ELSIF Failed OR (NOT Busy AND Done) THEN
	F_SetpointEnableExecute := FALSE;
ELSE
	// e.g. the request ended while the block is still busy: keep Execute until it is done
	F_SetpointEnableExecute := Execute;
END_IF

END_FUNCTION

// ---- POUs/FB_Axis.TcPOU
FUNCTION_BLOCK FB_Axis
VAR_INPUT
	// enable the axis
	Enable:		BOOL;
	// reset the axis after error
	Reset: 		BOOL;
	// Move the Axis to a given position
	MoveAxis: 	BOOL;
	// HomeAxis;
	HomeAxis:	BOOL;
	// Stop the axis
	StopAxis:	BOOL;
	// position to move to
	Position: 	LREAL;
	// maximum velocity
	Velocity:	LREAL := 10.0;
	// expected average tracking velocity
	TrackVelocityRef: LREAL := 0.0;
	// Tracking direction (-1,0,1)
	TrackDirectionRef: INT := 0;
	// PosDiff for isTracking (arcsec)
	TrackEnvelope: LREAL := 5.0;
	// Enable movement in positive direction (considering limit switch)
	Enable_Positive:	BOOL := TRUE;
	// Enable movement in negative direction (considering limit switch)
	Enable_Negative:	BOOL := TRUE;
	// jog forward
	Jog_Forward:		BOOL := FALSE;
	// jog backward
	Jog_Backwards:		BOOL := FALSE;
	// calibration input for homing
	bCalibrationCam:	BOOL;
	isModuloAxis:		BOOL := FALSE;
	// enable external setpoint generator
	Tracking:			BOOL;
	HomingMode:			MC_HomingMode := MC_HomingMode.MC_DefaultHoming;
END_VAR
VAR_OUTPUT
	// Reset has been executed
	ResetDone:	BOOL;
	// the axis is in target position
	MoveDone:	BOOL;
	// the axis hass jogged
	JogDone:	BOOL;
	// the axis has stopped
	StopDone: 	BOOL;
	// the axis was calibrated and has come to a standstill
	HomeDone:	BOOL;
	// the axis is ready
	Ready:		BOOL;
	// the command has been aborted
	CommandAborted: BOOL;
	// axis busy
	Busy: 		BOOL;
	// axis is moving
	Active: 	BOOL;
	// axis is stopping
	Stopping:	BOOL;
	// axis is standing still (no commands issued) this should be the default
	StandStill:	BOOL;
	// axis is in motion
	InMotion:	BOOL;
	// axis is homing
	Homing:		BOOL;
	// axis is Accelerating or Decelerating
	InRamp:		BOOL;
	// axis is tracking on position
	isTracking:	BOOL;
	//	error condition
	Error: 		BOOL;
	// number of error
	ErrorID: 	UDINT;
	// actual position of the axis
	ActualPosition: LREAL;
	// axis is calibrated;
	Calibrated:	BOOL := FALSE;

END_VAR
VAR
	Axis_Power:		MC_Power;
	Axis_Reset:		MC_Reset;
	Axis_Move:		MC_MoveAbsolute;
	Axis_Modulo:	MC_MoveModulo;
	//Axis_Position:	MC_ReadActualPosition;
	Axis_Stop:		MC_Stop;
	Axis_Status:	MC_ReadStatus;
	Axis_Home:		MC_Home;
	Axis_Jog: 		MC_Jog;
	Axis_SetpointEnable:	MC_ExtSetPointGenEnable;
	SetpointEnableFailed:	BOOL;	// setpoint enable failed; no retry until Reset or the end of the track request (#9)
	Axis_SetpointDisable:	MC_ExtSetPointGenDisable;
	StopAllowed:	BOOL;
	// Direction for Axis_SetpointFeed
	Direction:			DINT;
	// difference between set position and measured position
	PositionDifference:	LREAL;
	TrackPosition:		LREAL;
	TrackVelocity:		LREAL;
	TrackAcceleration:	LREAL;
END_VAR

VAR_IN_OUT
	// axis reference
	AxisRef:	AXIS_REF;
END_VAR

// query the status of the axis at the beginning of the cycle
Axis_Status(Enable := TRUE,
			Axis := AxisRef);

// Enable the axis (power signal or manual enable)
Axis_Power(
	Axis := AxisRef,
	Enable := Enable,
	Enable_Positive := Enable_Positive,
	Enable_Negative := Enable_Negative,
	Override := 100.0,
	Status => Ready);

Axis_Reset(
	Axis := 	AxisRef,
	Execute := 	Reset,
	Done => 	ResetDone);

(* Tracking section ********************************************** *)

IF Tracking THEN
	PositionDifference := Position - ActualPosition;
	TrackPosition := Position;
	IF ABS(PositionDifference) > 0.01 THEN
		TrackVelocity := 0.05;
		TrackAcceleration := 0.05;
	ELSE
		TrackAcceleration := 0.005;
	END_IF
ELSE
	TrackPosition := ActualPosition;
	TrackVelocity := 0.0;
	TrackAcceleration := 0.0;
END_IF


IF NOT Tracking OR ABS(PositionDifference) < 1E-5 THEN
	Direction := TrackDirectionRef;
	TrackAcceleration := 0.005;
ELSIF PositionDifference < 0.0 THEN
	Direction := -1;
	IF TrackDirectionRef = -1 THEN
		TrackVelocity := ABS(LIMIT(0.0, Velocity, 0.009));
	ELSE
		TrackVelocity := ABS(LIMIT(0.0, Velocity-TrackVelocityRef, 0.009));
	END_IF

ELSE
	Direction := 1;
	IF TrackDirectionRef = 1 THEN
		TrackVelocity := ABS(LIMIT(0.0, Velocity, 0.009));
	ELSE
		TrackVelocity := ABS(LIMIT(0.0, Velocity-TrackVelocityRef, 0.009));
	END_IF
END_IF



isTracking := Tracking AND ABS(Position - ActualPosition) < (TrackEnvelope/3600.0);
// drops Execute on an error and re-arms on Reset or a new track request (#9), see F_SetpointEnableExecute
Axis_SetpointEnable.Execute := F_SetpointEnableExecute(
	Request :=	Tracking AND Ready AND Calibrated AND NOT StopAxis,
	Tracking :=	Tracking,
	Reset :=	Reset,
	Execute :=	Axis_SetpointEnable.Execute,
	Busy :=		Axis_SetpointEnable.Busy,
	Done :=		Axis_SetpointEnable.Done,
	Error :=	Axis_SetpointEnable.Error,
	Failed :=	SetpointEnableFailed);

Axis_SetpointEnable(Axis := AxisRef,
	Position :=		TrackPosition,	// final destination
	PositionType := POSITIONTYPE_ABSOLUTE);

MC_ExtSetPointGenFeed(
	Position :=		TrackPosition,
	Velocity :=		Direction*TrackVelocity,
	Acceleration :=	TrackAcceleration,
	Direction :=	Direction,
	Axis :=			AxisRef);

Axis_SetpointDisable(Axis := AxisRef,
	Execute := NOT Tracking);

(* end of tracking section  ********************************************** *)

IF isModuloAxis THEN
	Axis_Modulo(
		Axis := 		AxisRef,
		Execute := 		MoveAxis AND Ready AND Calibrated,
		Position := 	Position,
		Velocity :=		Velocity,
		Direction := 	MC_Shortest_Way,
		Done => 		MoveDone);
ELSE
	Axis_Move(
		Axis := 		AxisRef,
		Execute := 		MoveAxis AND Ready AND Calibrated,
		Position := 	Position,
		Velocity := 	Velocity,
		Done => 		MoveDone);
END_IF

Axis_Jog(
	JogForward := 	Jog_Forward AND Ready AND Enable_Positive,
	JogBackwards := Jog_Backwards AND Ready AND Enable_Negative,
	Mode := 		MC_JOGMODE_STANDARD_FAST,
	Done => 		JogDone,
	Axis := 		AxisRef);


Axis_Home(
	Axis := 			AxisRef,
	Execute := 			HomeAxis AND Ready,
	// NOTE: the reference position is the Position input (also the MoveAxis target), not a separate
	// home position. HalfBROT and the IAG50cm focus axis rely on this (they set Position to the
	// calibration position before homing), so do not change without migrating callers.
	Position := 		Position,
	HomingMode :=		HomingMode,
	bCalibrationCam := 	bCalibrationCam,
	Done => 			HomeDone);

(*
IF (MoveDone OR HomeDone OR JogDone) AND NOT Axis_Status.StandStill THEN
	StopAxis := TRUE;
END_IF
*)
IF MoveDone AND NOT Axis_Modulo.Busy AND NOT Axis_Move.Busy THEN
	MoveAxis := FALSE;
END_IF

IF JogDone THEN
	Jog_Forward := FALSE;
	Jog_Backwards := FALSE;
END_IF

IF Axis_Status.Status.Homed THEN
	Calibrated := TRUE;
	// NOTE: HomeDone is a level (TRUE while the axis is homed), not a one-cycle pulse; IAG50cm's
	// FB_HourAngleControl/FB_DeclinationControl combine it with FB_LatchHome.Done. Use Calibrated.
	HomeDone := TRUE;
	// do not cancel a re-home request in the cycle it starts on an already-homed axis
	IF NOT Axis_Home.Busy THEN
		HomeAxis := FALSE;
	END_IF
ELSE
	Calibrated := FALSE;
	HomeDone := FALSE;
END_IF

IF StopDone THEN
	StopAxis := FALSE;
END_IF

StopAllowed :=	Axis_Status.StandStill OR
				Axis_Status.ContinuousMotion OR
				Axis_Status.DiscreteMotion OR
				Axis_Status.SynchronizedMotion OR
				Axis_Status.Homing;

Axis_Stop(
	Axis := 	AxisRef,
	Execute := 	StopAxis AND StopAllowed,
	Done => 	StopDone);
(*
Axis_Position(
	Axis := 	AxisRef,
	Enable := 	Calibrated,
	Position => AbsolutePosition);
*)
IF isModuloAxis THEN
	ActualPosition := AxisRef.NcToPlc.ModuloActPos; // required e.g. for Filterwheel
ELSE
	ActualPosition := AxisRef.NcToPlc.ActPos;
END_IF

IF Axis_Power.Error THEN
	ErrorID := Axis_Power.ErrorID;
END_IF

IF Axis_SetpointEnable.Error THEN
	ErrorID := Axis_SetpointEnable.ErrorID;
END_IF

IF Axis_Reset.Error THEN
	ErrorID := Axis_Reset.ErrorID;
END_IF

IF Axis_Modulo.Error THEN
	ErrorID := Axis_Modulo.ErrorID;
END_IF

IF Axis_Move.Error THEN
	ErrorID := Axis_Move.ErrorID;
END_IF

IF Axis_Home.Error THEN
	ErrorID := Axis_Home.ErrorID;
END_IF

IF Axis_Jog.Error THEN
	ErrorID := Axis_Jog.ErrorID;
END_IF

IF Axis_Stop.Error THEN
	ErrorID := Axis_Stop.ErrorID;
END_IF

IF Axis_Status.Error THEN
	ErrorID := Axis_Status.ErrorID;
END_IF
Busy := 	Axis_SetpointEnable.Busy OR
			Axis_Reset.Busy OR
			Axis_Modulo.Busy OR
			Axis_Move.Busy OR
			Axis_Home.Busy OR
			Axis_Jog.Busy;

Error := 	Axis_Power.Error OR
			Axis_SetpointEnable.Error OR
			SetpointEnableFailed OR		// keeps a setpoint enable error visible after Execute dropped (#9)
			Axis_Reset.Error OR
			Axis_Modulo.Error OR
			Axis_Move.Error OR
			Axis_Home.Error OR
			Axis_Jog.Error OR
			Axis_Stop.Error OR
			Axis_Status.Error;

Active := 	// Axis_Power.Active OR //alsways true if enabled
			Axis_Modulo.Active OR
			Axis_Move.Active OR
			Axis_Home.Active OR
			Axis_Jog.Active OR
			Axis_Stop.Active;

CommandAborted :=	Axis_Modulo.CommandAborted OR
					Axis_Move.CommandAborted OR
					Axis_Home.CommandAborted OR
					Axis_Jog.CommandAborted OR
					Axis_Stop.CommandAborted;

IF NOT Error THEN
	ErrorID := 0;
END_IF

InMotion := Axis_Status.ConstantVelocity OR
			Axis_Status.DiscreteMotion OR
			Axis_Status.ContinuousMotion OR
			Axis_Status.SynchronizedMotion;
InRamp :=	Axis_Status.Accelerating OR
			Axis_Status.Decelerating;
Stopping := Axis_Status.Stopping;
StandStill := Axis_Status.StandStill;
Homing :=	Axis_Status.Homing;
// InPosition := AxisRef.NcToPlc.TargetPos;

END_FUNCTION_BLOCK

// ---- POUs/FB_BaseAxis.TcPOU
FUNCTION_BLOCK ABSTRACT FB_BaseAxis IMPLEMENTS I_BaseAxis
VAR_INPUT
	bEnable				: BOOL;		// enable the axis and its position control loop
	bReset				: BOOL;		// reset the axis
	bSoEReset			: BOOL;		// diagnostic reset
	bHomeAxis			: BOOL;		// Home the axis
	fPosition			: LREAL;	// position to move the axis to
	fVelocity			: LREAL;	// set the Velocity of the axis
	bMoveNeg			: BOOL;		// decrease position
	bMovePos			: BOOL;		// increase position
END_VAR
VAR_OUTPUT
	fActualPosition		: LREAL;	// actual_position of the axis
	bCalibrated			: BOOL;		// true if absolute calibration
	bError				: BOOL;		// true if error
	nErrorID			: UDINT;	// error ID of the axis
	bReady				: BOOL;		// drive is ready
END_VAR
VAR
	fbComm				: I_Comm;
	fbAxis				: FB_Axis;
	fbSoEReset			: FB_SoEReset;
	axisRef				: AXIS_REF;
END_VAR

PROPERTY ActualPosition : LREAL
GET
ActualPosition := fActualPosition;
END_GET
SET
fActualPosition := ActualPosition;
END_SET
END_PROPERTY

PROPERTY Busy : BOOL
GET
Busy := fbAxis.Busy;
END_GET
END_PROPERTY

PROPERTY Calibrated : BOOL
GET
Calibrated := bCalibrated;
END_GET
END_PROPERTY

PROPERTY Enable : BOOL
GET
Enable := bEnable;
END_GET
SET
bEnable := Enable;
END_SET
END_PROPERTY

PROPERTY Error : BOOL
GET
Error := bError;
END_GET
END_PROPERTY

PROPERTY ErrorID : UDINT
GET
ErrorID := nErrorID;
END_GET
END_PROPERTY

//FB_Init is always available implicitly and it is used primarily for initialization.
//The return value is not evaluated. For a specific influence, you can also declare the
//methods explicitly and provide additional code there with the standard initialization
//code. You can evaluate the return value.
METHOD FB_Init: BOOL
VAR_INPUT
    bInitRetains	: BOOL; // TRUE: the retain variables are initialized (reset warm / reset cold)
    bInCopyCode		: BOOL;  // TRUE: the instance will be copied to the copy code afterward (online change)
	comm			: I_Comm;   
END_VAR
THIS^.fbComm := comm;
END_METHOD

PROPERTY HomeAxis : BOOL
GET
HomeAxis := bHomeAxis;
END_GET
SET
bHomeAxis := HomeAxis;
END_SET
END_PROPERTY

PROPERTY InNegLimit : BOOL
GET
// no limit-switch input at this level; concrete subclasses must override this with a real
// hardware/soft-limit read. Left unoverridden, this always reports "not at the limit" -- the
// safe-looking value but not an accurate one (BROTLib#20)
InNegLimit := FALSE;
END_GET
END_PROPERTY

PROPERTY InPosLimit : BOOL
GET
// see InNegLimit -- same caveat, concrete subclasses must override with a real limit read
InPosLimit := FALSE;
END_GET
END_PROPERTY

PROPERTY isTracking : BOOL
GET
isTracking := fbAxis.isTracking;
END_GET
END_PROPERTY

PROPERTY MoveNeg : BOOL
GET
MoveNeg := bMoveNeg;
END_GET
SET
bMoveNeg := MoveNeg;
END_SET
END_PROPERTY

PROPERTY MovePos : BOOL
GET
MovePos := bMovePos;
END_GET
SET
bMovePos := MovePos;
END_SET
END_PROPERTY

PROPERTY Position : LREAL
GET
Position := fPosition;
END_GET
SET
fPosition := Position;
END_SET
END_PROPERTY

PROPERTY Ready : BOOL
GET
Ready := bReady;
END_GET
END_PROPERTY

METHOD Reset : BOOL
bReset := TRUE;
END_METHOD

PROPERTY Velocity : LREAL
GET
Velocity := fVelocity;
END_GET
SET
fVelocity := Velocity;
END_SET
END_PROPERTY

END_FUNCTION_BLOCK

// ---- POUs/FB_BLINK.TcPOU
FUNCTION_BLOCK FB_BLINK
VAR_INPUT
	blink:		E_Blink;
	ON_TIME:	TIME := T#500MS;
	OFF_TIME:	TIME := T#500MS;
END_VAR
VAR_OUTPUT
	Q:		BOOL;
END_VAR
VAR
    IMPULS   :TOF;
    PAUSE    :TOF;
END_VAR

CASE blink OF
	e_blink.slow:
		ON_TIME := T#500MS;
		OFF_TIME := T#500MS;
	e_blink.fast:
		ON_TIME := T#250MS;
		OFF_TIME := T#250MS;
	e_blink.short:
		ON_TIME := T#100MS;
		OFF_TIME := T#900MS;
	e_blink.long:
		ON_TIME := T#900MS;
		OFF_TIME := T#100MS;
END_CASE

IMPULS(IN:= NOT PAUSE.Q AND NOT IMPULS.Q, PT:= ON_TIME);
PAUSE(IN:= NOT PAUSE.Q AND NOT IMPULS.Q, PT:= OFF_TIME);
IF blink = e_blink.off THEN
	Q := FALSE;
ELSIF blink = e_blink.on THEN
	Q := TRUE;
ELSE
	Q := IMPULS.Q;	
END_IF

END_FUNCTION_BLOCK

// ---- POUs/FB_ButtonEnable.TcPOU
FUNCTION_BLOCK FB_ButtonEnable
VAR_INPUT
	SET:	BOOL;
	RESET:	BOOL;
END_VAR
VAR_IN_OUT
	Q: BOOL;
END_VAR
VAR
	trigger:	R_TRIG;
//	ftrigger:	F_TRIG;
END_VAR

trigger(CLK := SET);
//ftrigger(CLK := SET);

// if button was triggered, flip the state of the output
IF trigger.Q THEN
	Q := NOT Q;
END_IF

// if reset is enabled we disable the output
IF RESET THEN
	Q := FALSE;
END_IF

END_FUNCTION_BLOCK

// ---- POUs/FB_Horn.TcPOU
FUNCTION_BLOCK FB_Horn
VAR_INPUT
	horn:	E_Horn;
END_VAR
VAR_OUTPUT
		Q:		BOOL;
END_VAR
VAR
	ON_TIME:	TIME := T#500MS;
	OFF_TIME:	TIME := T#500MS;
	IMPULS   :TOF;
    PAUSE    :TOF;

END_VAR

CASE horn OF
	e_horn.off:
		ON_TIME := T#0MS;
		OFF_TIME := T#0MS;
	e_horn.beep:
		ON_TIME := T#500MS;
		OFF_TIME := T#500MS;
	e_horn.short:
		ON_TIME := T#3000MS;
		OFF_TIME := T#3000MS;
	e_horn.long:
		ON_TIME := T#5000MS;
		OFF_TIME := T#5000MS;
END_CASE

// same IMPULS/PAUSE oscillator as FB_BLINK: PAUSE must actually run for the pair
// to alternate ON_TIME/OFF_TIME -- without it (the previous bug) NOT PAUSE.Q is
// always TRUE and IMPULS just retriggers itself every cycle, i.e. stays on
IMPULS(IN:= NOT PAUSE.Q AND NOT IMPULS.Q, PT:= ON_TIME);
PAUSE(IN:= NOT PAUSE.Q AND NOT IMPULS.Q, PT:= OFF_TIME);
IF horn = e_horn.off THEN
	Q := FALSE;
ELSE
	Q := IMPULS.Q;
END_IF

END_FUNCTION_BLOCK

// ---- POUs/FB_TONTP.TcPOU
FUNCTION_BLOCK FB_TONTP
VAR_INPUT
	IN :	BOOL;
	 PT1:	TIME := T#1000MS;
	 PT2:	TIME := T#1000MS;
END_VAR
VAR_OUTPUT
	Q:	BOOL;
END_VAR
VAR
	ton:	TON;
	tp:		TP;
END_VAR

ton(IN := IN, PT := PT1);
tp(IN := ton.Q, PT := PT2, Q => Q);

END_FUNCTION_BLOCK

// ---- POUs/F_YREAL.TcPOU
FUNCTION F_YREAL : REAL
VAR_INPUT
	fX:		LREAL;
	fXmin:	REAL := 0.0;
	fXmax:	REAL := 32767.0;
	fYmin:	REAL := 0.0;
	fYmax:	REAL := 1.0;
	cut:    BOOL := TRUE;
END_VAR
VAR
	fgain:		LREAL;
	foffset:	LREAL;
END_VAR

(*
y = mx+b

		    delta Y	  fYmax - fYmin
m = fgain = ------- = -------------
			delta X	  fXmax - fXmin

b = foffset = y - m*x = y - fgain*x
					  = fYmin - fgain * fXmin
*)

// y = fgain * x + foffset

IF (fXmax - fXmin) <> 0 THEN

	// Berechnung der Steigung
	fgain := (fYmax - fYmin) / (fXmax - fXmin);

	// Berechnung des Offsets
	foffset := fYmin - (fgain * fXmin);

	// Berechnung von F_Y

	F_YREAL := LREAL_TO_REAL(fgain * fX + foffset);
	IF cut THEN
		// LIMIT(MN, IN, MX) requires MN <= MX; fYmin/fYmax can be given inverted
		// (e.g. mapping onto a descending range), so clamp against the actual
		// low/high bound instead of assuming fYmin is the low one
		F_YREAL := LIMIT(MIN(fYmin, fYmax), F_YREAL, MAX(fYmin, fYmax));
	END_IF
END_IF

END_FUNCTION

// ---- POUs/NCError_TO_STRING.TcPOU
FUNCTION NCError_TO_STRING : STRING(255)
VAR_INPUT
	// NC Error ID
	ErrorID:	UDINT;
END_VAR
VAR
END_VAR

NCError_TO_STRING := '';

CASE ErrorID OF
	16#D012:	NCError_TO_STRING := 'Control and power section ready (no error)';
	16#D013:	NCError_TO_STRING := 'Axis in operation (no error)';
	16#4220:	NCError_TO_STRING := 'Group not ready / group not ready for new task';
	16#4253:	NCError_TO_STRING := 'Reference cam became free too soon';
	16#4257:	NCError_TO_STRING := 'Function not allowed';
	16#4260:	NCError_TO_STRING := 'Controller enable';
	16#42EF:	NCError_TO_STRING := 'Axis is locked for motion commands because a stop command is still active';
	16#4466:	NCError_TO_STRING := 'Invalid IO data FOR more than n subsequent NC cycles (encoder)';
	16#4550: 	NCError_TO_STRING := 'Following error monitoring (position)';
	16#4650:	NCError_TO_STRING := 'Drive hardware not ready to operate';
	16#4B07:	NCError_TO_STRING := 'Timeout axis function block';
	16#4B09:	NCError_TO_STRING := 'Axis is not ready';
	16#4B0A:	NCError_TO_STRING := 'Error during referencing';
	16#ECD0:	NCError_TO_STRING := 'Positive limit switch warning.';				
	16#ED43:	NCError_TO_STRING := 'Under-voltage - DC link.';				
	16#F324:	NCError_TO_STRING := 'Excessive position command value deviation';				
	16#F601:	NCError_TO_STRING := 'Calibrate commutation offset error.';				

ELSE
	NCError_TO_STRING := DWORD_TO_HEXSTR(ErrorID, 4, FALSE);
END_CASE

END_FUNCTION

// ---- POUs/Pointing/FB_PointingModelForward.TcPOU
FUNCTION_BLOCK FB_PointingModelForward
VAR_INPUT
	fAzimuth		: LREAL;	// current azimuth of telescope in degrees
	fElevation		: LREAL;	// current elevation of telescope in degrees
END_VAR
VAR_OUTPUT
	fAzimuthOffset	: LREAL;	// calculated azimuth offset of telescope in degrees
	fElevationOffset	: LREAL;	// calculated elevation offset of telescope in degrees
END_VAR
VAR
	AOFF			: LREAL := 0.0;		// azimuth encoder zero offset
	BNP				: LREAL := 0.0;		// collimation error of the electromagnetic axis
	AN_A			: LREAL := 0.0;		// azimuth axis offset/misalignment north-south
	AE_A			: LREAL := 0.0;		// azimuth axis offset/misalignment east-west,
	NPAE			: LREAL := 0.0;		// Non-perpendicularity between the mount azimuth and elevation axes	
	
	EOFF			: LREAL := 0.0;		// elevation encoder zero offset
	AN_E			: LREAL := 0.0;		// azimuth axis offset/misalignment north-south
	AE_E			: LREAL := 0.0;		// azimuth axis offset/misalignment east-west
	TF				: LREAL := 0.0;		// gravitational flexure correction at the horizon	
	
	fTanElevation	: LREAL;
	fCosElevation	: LREAL;
END_VAR

IF fElevation<89.9 THEN
	fTanElevation := TAN(fElevation * GVL_Math.d2r);
	fCosElevation := COS(fElevation * GVL_Math.d2r);
ELSE // clamp values so that we do not run into DIV by zero or overflow
	fTanElevation := 572.9572133543033;
	fCosElevation := 0.0017453283658982613;
END_IF

//d(az)=AOFF-BNP/cos(el)+NPAE*tan(el)+AAN*sin(az)*tan(el)-AAE*cos(az)*tan(el)
fAzimuthOffset := AOFF - BNP/fCosElevation + AN_A*SIN(fAzimuth * GVL_Math.d2r)*fTanElevation - AE_A*COS(fAzimuth * GVL_Math.d2r)*fTanElevation + NPAE*fTanElevation;
fElevationOffset := EOFF + AN_E*COS(fAzimuth * GVL_Math.d2r) + AE_E*SIN(fAzimuth * GVL_Math.d2r) + TF*COS(fElevation * GVL_Math.d2r);

METHOD FB_init : BOOL
VAR_INPUT
	bInitRetains : BOOL; // if TRUE, the retain variables are initialized (warm start / cold start)
	bInCopyCode : BOOL;  // if TRUE, the instance afterwards gets moved into the copy code (online change)
	
	AOFF			: LREAL := 0.0;		// azimuth encoder zero offset
	BNP				: LREAL := 0.0;		// collimation error of the electromagnetic axis
	AN_A			: LREAL := 0.0;		// azimuth axis offset/misalignment north-south
	AE_A			: LREAL := 0.0;		// azimuth axis offset/misalignment east-west,
	NPAE			: LREAL := 0.0;		// Non-perpendicularity between the mount azimuth and elevation axes	
	
	EOFF			: LREAL := 0.0;		// elevation encoder zero offset
	AN_E			: LREAL := 0.0;		// azimuth axis offset/misalignment north-south
	AE_E			: LREAL := 0.0;		// azimuth axis offset/misalignment east-west
	TF				: LREAL := 0.0;		// gravitational flexure correction at the horizon		
END_VAR
THIS^.AOFF := AOFF;
THIS^.BNP  := BNP;
THIS^.AN_A := AN_A;
THIS^.AE_A := AE_A;
THIS^.NPAE := NPAE;
THIS^.EOFF := EOFF;
THIS^.AN_E := AN_E;
THIS^.AE_E := AE_E;
THIS^.TF   := TF;
END_METHOD

END_FUNCTION_BLOCK

// ---- POUs/Pointing/FB_PointingModelInversion.TcPOU
FUNCTION_BLOCK FB_PointingModelInversion
VAR_INPUT
	fAzimuth		: LREAL;	// current azimuth of telescope in degrees
	fElevation		: LREAL;		// current elevation of telescope in degrees
END_VAR
VAR_OUTPUT
	fAzimuthOffset		: LREAL;	// calculated azimuth offset of telescope in degrees
	fElevationOffset	: LREAL;	// calculated elevation offset of telescope in degrees
END_VAR
VAR
	i				: UINT;
	d_el			: LREAL := 0.0;
	d_az			: LREAL := 0.0;
	fElevationClamped	: LREAL;
	fbPointing		: REFERENCE TO FB_PointingModelForward;
END_VAR

d_el := 0.0;
d_az := 0.0;

// fbPointing is only ever set via FB_init(fbPointing := ...); nothing enforces that a consumer
// actually does, and calling through an unassigned REFERENCE TO crashes the whole PLC task (#7).
// Leave the offsets at 0.0 (no correction) rather than crash.
IF NOT __ISVALIDREF(fbPointing) THEN
	fAzimuthOffset := 0.0;
	fElevationOffset := 0.0;
	RETURN;
END_IF

// FB_PointingModelForward's own BNP/cos(el) term grows without bound approaching the zenith (89.9 deg is
// where the forward model switches to its own fixed clamp); feeding the iteration an elevation past that
// point keeps growing the offset further instead of converging to the bounded value the forward model
// would give at 89.9 deg
fElevationClamped := MIN(fElevation, 89.9);

// 2 passes converge to < 0.1" for every elevation/coefficient combination tried; 5 keeps a wide margin
// (needed for BROTLibTests' Inversion_Round_Trip, which checks self-consistency to 1e-9 deg)
FOR i:=0 TO 4 BY 1 DO
	fbPointing(
		fAzimuth   		 := fAzimuth   		  - d_az,
		fElevation 		 := fElevationClamped - d_el,
		fAzimuthOffset   => d_az,
		fElevationOffset => d_el,
	);
END_FOR;

fAzimuthOffset   := d_az;
fElevationOffset := d_el;

METHOD FB_init : BOOL
VAR_INPUT
	bInitRetains : BOOL; // if TRUE, the retain variables are initialized (warm start / cold start)
	bInCopyCode : BOOL;  // if TRUE, the instance afterwards gets moved into the copy code (online change)
	
	fbPointing		: REFERENCE TO FB_PointingModelForward;
END_VAR
THIS^.fbPointing REF= fbPointing;
END_METHOD

END_FUNCTION_BLOCK

// ---- POUs/Tracking/F_Azimuthvelocity.TcPOU
FUNCTION F_Azimuthvelocity : LREAL
VAR_INPUT
	// elevation in degrees
	elevation: 	LREAL;
	// azimuth in degrees
	azimuth:	LREAL;
	// observers latitude in degrees
	latitude:	LREAL;
END_VAR
VAR
END_VAR

IF ABS(COS(elevation * GVL_Math.d2r))> 1.0e-3 THEN
	F_Azimuthvelocity := (SIN(latitude * GVL_Math.d2r) - COS(latitude * GVL_Math.d2r) * COS(azimuth * GVL_Math.d2r) * TAN(elevation * GVL_Math.d2r))* GVL_Math.Omega;
ELSE
	F_Azimuthvelocity := 0.0;	
END_IF

END_FUNCTION

// ---- POUs/Tracking/F_DerotatorPosition2.TcPOU
FUNCTION F_DerotatorPosition2 : LREAL
VAR_INPUT
	// azimuth of the target
	azimuth: LREAL;
	// elevation of the target in degrees
	elevation: LREAL;
	// latitude in degrees
	latitude:	LREAL;
	// sign for elevation
	sign:	LREAL := 1.0;
END_VAR
VAR
	// parallactic angle
	az, el, la: LREAL;
	parallactic_angle:	LREAL;
	//zenith_distance: LREAL;
END_VAR
VAR CONSTANT
	//h2r:	LREAL := PI/12.0;
	//h2d:	LREAL := 15.0;
END_VAR

// calculate the parallactic angle
az := MODABS(azimuth, 360.0) * GVL_Math.d2r;
el := LIMIT(0.0, elevation, 90.0) * GVL_Math.d2r;
la := LIMIT(-90.0, latitude, 90.0) * GVL_Math.d2r;

parallactic_angle := - GVL_Math.r2d * ATAN2(SIN(az), TAN(la)*COS(el)-SIN(el)*COS(az));

// use the same clamped elevation as the trigonometry above, not the raw input
F_DerotatorPosition2 := parallactic_angle - sign * (el * GVL_Math.r2d);
F_DerotatorPosition2 := MODABS(F_DerotatorPosition2, 360.0);

END_FUNCTION

// ---- POUs/Tracking/F_Derotatorvelocity.TcPOU
FUNCTION F_Derotatorvelocity : LREAL
VAR_INPUT
	// azimuth in degrees
	azimuth:	LREAL;
	// elevation in degrees
	elevation: 	LREAL;
	// observers latitude in degrees
	latitude:	LREAL;
	// sign for elevation, must match the sign passed to F_DerotatorPosition2
	sign:	LREAL := 1.0;
END_VAR
VAR
END_VAR

(*
source: https://github.com/cytan299/field_derotator/blob/master/field_derotator_formula/field_derotator_formula.pdf
https://circuitcellar.com/research-design-hub/projects/field-derotator-for-astrophotography-part-1/

returns the rotational velocity for the de-rotator in degrees per second
azimuth, latitutde and elevation are converted to radians
*)
IF ABS(COS(elevation * GVL_Math.d2r))> 1.0e-3 THEN
	// this closed form is the parallactic-angle rate minus the elevation rate (i.e. the sign = 1
	// case of F_DerotatorPosition2); (1 - sign) * elevation rate corrects it for any other sign
	F_Derotatorvelocity := -GVL_Math.Omega * COS(azimuth * GVL_Math.d2r) * COS(latitude * GVL_Math.d2r) / COS(elevation * GVL_Math.d2r)  - GVL_Math.Omega *COS(latitude * GVL_Math.d2r) * SIN(azimuth * GVL_Math.d2r)
		+ (1.0 - sign) * F_Elevationvelocity(azimuth, latitude);
ELSE
	F_Derotatorvelocity := 0.0;
END_IF

END_FUNCTION

// ---- POUs/Tracking/F_Elevationvelocity.TcPOU
FUNCTION F_Elevationvelocity : LREAL
VAR_INPUT
	// azimuth in degrees
	azimuth:	LREAL;
	// observers latitude in degrees
	latitude:	LREAL;
END_VAR
VAR
END_VAR

//returns the rotational velocity for the azimuth in degrees per second
F_Elevationvelocity := SIN(azimuth*GVL_Math.d2r) * COS(latitude*GVL_Math.d2r) * GVL_Math.Omega;

END_FUNCTION

// ---- Telescope/FB_AltAzTelescopeControl.TcPOU
FUNCTION_BLOCK ABSTRACT FB_AltAzTelescopeControl EXTENDS FB_BaseTelescopeControl IMPLEMENTS I_AltAzTelescope
VAR_INPUT
	fElevationOffset	: LREAL := 0.0;		// absolute offset for elevation
	fAzimuthOffset 		: LREAL := 0.0;		// absolute offset for azimuth
	fDerotatorOffset	: LREAL := 0.0;		// offset for the de-rotator
	// UT1-UTC (seconds, IERS). 0.0 = treat UTC as UT1 (no correction), matching FB_EQ2HOR/
	// FB_HOR2EQ's own default. Set via MQTT by an external time bridge (Dut1 property, see
	// FB_Comm_MQTT_Influx); reverts to 0.0 if nothing fresh arrives for a while (below).
	fDut1				: LREAL := 0.0;
END_VAR
VAR_OUTPUT
	fDerotatorCurrent	: LREAL;	// current position in derotator (calculated) (without pointing and offset correction)
END_VAR
VAR
	eq2hor				: FB_EQ2HOR;
	hor2eq				: FB_HOR2EQ;

	fDerotatorCalc		: LREAL;	// derotator angle calcuilated

	bDut1Received		: BOOL;
	tonDut1Stale		: TON := (PT := T#10M);
END_VAR
// The pointing-model coefficients live in FB_PointingModelForward, set by the caller (#10).

SUPER^();

METHOD _PublishTelemetry : BOOL
VAR_INPUT
END_VAR
SUPER^._PublishTelemetry();

fbComm.Publish('telescope', 'dome', 'POSITION.INSTRUMENTAL.AZ.OFFSET', LREAL_TO_STRING(fAzimuthOffset));
fbComm.Publish('telescope', 'dome', 'POSITION.INSTRUMENTAL.ALT.OFFSET', LREAL_TO_STRING(fElevationOffset));
END_METHOD

PROPERTY AltitudeOffset : LREAL
GET
AltitudeOffset := THIS^.fElevationOffset;
END_GET
SET
THIS^.fElevationOffset := AltitudeOffset;
END_SET
END_PROPERTY

PROPERTY AzimuthOffset : LREAL
GET
AzimuthOffset := THIS^.fAzimuthOffset;
END_GET
SET
THIS^.fAzimuthOffset := AzimuthOffset;
END_SET
END_PROPERTY

PROPERTY DerotatorOffset : LREAL
GET
DerotatorOffset := THIS^.fDerotatorOffset;
END_GET
SET
THIS^.fDerotatorOffset := DerotatorOffset;
END_SET
END_PROPERTY

PROPERTY Dut1 : LREAL
GET
Dut1 := THIS^.fDut1;
END_GET
SET
THIS^.fDut1 := Dut1;
THIS^.bDut1Received := TRUE;
END_SET
END_PROPERTY

END_FUNCTION_BLOCK

// ---- Telescope/FB_RaDecTelescopeControl.TcPOU
FUNCTION_BLOCK FB_RaDecTelescopeControl EXTENDS FB_BaseTelescopeControl IMPLEMENTS I_RaDecTelescope;
VAR_INPUT
END_VAR
VAR_OUTPUT
END_VAR
VAR
	eq2hor				: FB_EQ2HOR;
	hor2eq				: FB_HOR2EQ;

	fHourAngleOffset	: LREAL := 0.0;		// absolute offset for hour angle
	fDeclinationOffset	: LREAL := 0.0;		// absolute offset for declination
	
	fHourAngleVelocity	: LREAL;	// rotational velocity of the HA
	fDeclinationVelocity: LREAL;	// rotational velocity of the declination
	
	fElevationPointing  	: LREAL;	// true position of the elevation with applied pointing model
	fAzimuthPointing    	: LREAL;	// true position of the azimuth with applied pointing model
	fRightAscensionPointing	: LREAL;	// RA from pointing Az/El
	fDeclinationPointing	: LREAL;	// Dec from pointing Az/El
	
	fDerotationSign	: LREAL := 1.0;	// sign of derotation
END_VAR
VAR PERSISTENT
	EOFF				: LREAL;	// elevation encoder zero offset
	AN_E				: LREAL;	// azimuth axis offset/misalignment north-south
	AE_E				: LREAL;	// azimuth axis offset/misalignment east-west
	TF					: LREAL;	// gravitational flexure correction at the horizon
	AOFF				: LREAL;	// azimuth encoder zero offset
	BNP					: LREAL;	// collimation error of the electromagnetic axis
	AN_A				: LREAL;	// azimuth axis offset/misalignment north-south
	AE_A				: LREAL;	// azimuth axis offset/misalignment east-west,
	NPAE				: LREAL;	// Non-perpendicularity between the mount azimuth and elevation axes
END_VAR

SUPER^();

// Alt/Az to RA/Dec
hor2eq(alt := fElevation, 
		az := fAzimuth,
		jd := fJD,
		lat := telescopeConfig.latitude,
		lon := telescopeConfig.longitude,
		altitude := telescopeConfig.altitude,
		ra => fRightAscensionCalc,
		dec => fDeclinationCalc);
		
// to HA
fHourAngleCalc := 0.0;

// apply pointing model
//fRightAscensionCalc := fRightAscensionCalc + PointingModelRightAscension
//fDeclinationCalc := fDeclinationCalc + PointingModelDeclination 

// calculate velocities
//fHourAngleVelocity := F_Elevationvelocity(fAzimuthCalc, telescopeConfig.latitude);
//fDeclinationVelocity := F_Azimuthvelocity(fElevationCalc, fAzimuthCalc, telescopeConfig.latitude);

// apply reverse pointing model
//fElevationPointing := fElevationCurrent - PointingModelElevation(fAzimuthCurrent, fElevationCurrent, EOFF, AN_E, AE_E, TF);
//fAzimuthPointing := fAzimuthCurrent - PointingModelAzimuth(fAzimuthCurrent, fElevationCurrent, AOFF, BNP, AN_A, AE_A, NPAE);

// add offsets
//fElevationCurrent := fElevationPointing - fElevationOffset;
//fAzimuthCurrent := fAzimuthPointing - fAzimuthOffset;

